REGION Network 52: Call CM Electrode Fix Left Top Up/Down (LBC_TwoWayActuator)
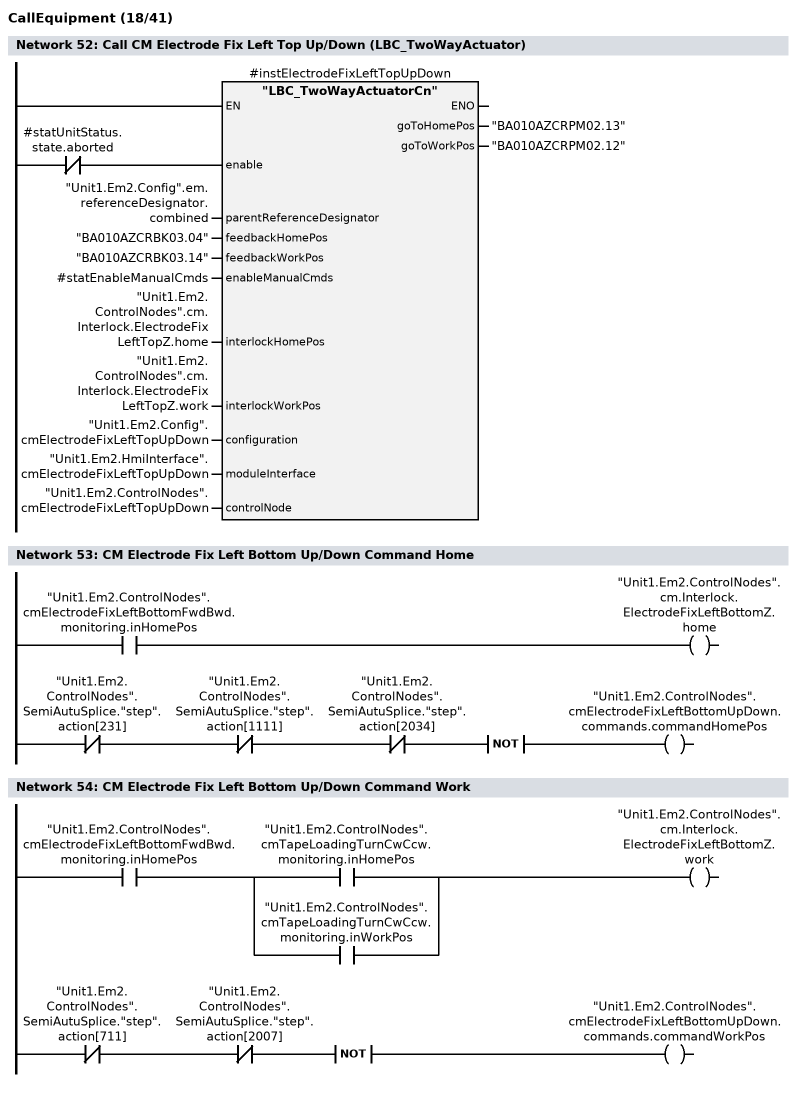
   RUNG wire#powerrail
      #instElectrodeFixLeftTopUpDown(enable := wire#w1, parentReferenceDesignator := "Unit1.Em2.Config".em.referenceDesignator.combined, feedbackHomePos := "BA010AZCRBK03.04", feedbackWorkPos := "BA010AZCRBK03.14", enableManualCmds := #statEnableManualCmds, interlockHomePos := "Unit1.Em2.ControlNodes".cm.Interlock.ElectrodeFixLeftTopZ.home, interlockWorkPos := "Unit1.Em2.ControlNodes".cm.Interlock.ElectrodeFixLeftTopZ.work, configuration := "Unit1.Em2.Config".cmElectrodeFixLeftTopUpDown, moduleInterface := "Unit1.Em2.HmiInterface".cmElectrodeFixLeftTopUpDown, controlNode := "Unit1.Em2.ControlNodes".cmElectrodeFixLeftTopUpDown, goToHomePos => "BA010AZCRPM02.13", goToWorkPos => "BA010AZCRPM02.12")
   END_RUNG
   RUNG wire#powerrail
      I_Contact( #statUnitStatus.state.aborted )
   END_RUNG wire#w1
   // the same network as SCL:
   #instElectrodeFixLeftTopUpDown(enable := NOT #statUnitStatus.state.aborted,   // "LBC_TwoWayActuatorCn"
                           parentReferenceDesignator := "Unit1.Em2.Config".em.referenceDesignator.combined,
                           feedbackHomePos := "BA010AZCRBK03.04",
                           feedbackWorkPos := "BA010AZCRBK03.14",
                           enableManualCmds := #statEnableManualCmds,
                           interlockHomePos := "Unit1.Em2.ControlNodes".cm.Interlock.ElectrodeFixLeftTopZ.home,
                           interlockWorkPos := "Unit1.Em2.ControlNodes".cm.Interlock.ElectrodeFixLeftTopZ.work,
                           configuration := "Unit1.Em2.Config".cmElectrodeFixLeftTopUpDown,
                           moduleInterface := "Unit1.Em2.HmiInterface".cmElectrodeFixLeftTopUpDown,
                           controlNode := "Unit1.Em2.ControlNodes".cmElectrodeFixLeftTopUpDown,
                           goToHomePos => "BA010AZCRPM02.13",
                           goToWorkPos => "BA010AZCRPM02.12");
END_REGION

REGION Network 53: CM Electrode Fix Left Bottom Up/Down Command Home
   RUNG wire#powerrail
      Contact( "Unit1.Em2.ControlNodes".cmElectrodeFixLeftBottomFwdBwd.monitoring.inHomePos )
      Coil( "Unit1.Em2.ControlNodes".cm.Interlock.ElectrodeFixLeftBottomZ.home )
   END_RUNG
   RUNG wire#powerrail
      I_Contact( "Unit1.Em2.ControlNodes".SemiAutuSplice."step".action[231] )
      I_Contact( "Unit1.Em2.ControlNodes".SemiAutuSplice."step".action[1111] )
      I_Contact( "Unit1.Em2.ControlNodes".SemiAutuSplice."step".action[2034] )
      Not()
      Coil( "Unit1.Em2.ControlNodes".cmElectrodeFixLeftBottomUpDown.commands.commandHomePos )
   END_RUNG
   // the same network as SCL:
   "Unit1.Em2.ControlNodes".cm.Interlock.ElectrodeFixLeftBottomZ.home := "Unit1.Em2.ControlNodes".cmElectrodeFixLeftBottomFwdBwd.monitoring.inHomePos;
   "Unit1.Em2.ControlNodes".cmElectrodeFixLeftBottomUpDown.commands.commandHomePos := NOT (NOT "Unit1.Em2.ControlNodes".SemiAutuSplice."step".action[231] AND NOT "Unit1.Em2.ControlNodes".SemiAutuSplice."step".action[1111] AND NOT "Unit1.Em2.ControlNodes".SemiAutuSplice."step".action[2034]);
END_REGION

REGION Network 54: CM Electrode Fix Left Bottom Up/Down Command Work
   RUNG wire#powerrail
      Contact( "Unit1.Em2.ControlNodes".cmElectrodeFixLeftBottomFwdBwd.monitoring.inHomePos )
      wire#w1
      Contact( "Unit1.Em2.ControlNodes".cmTapeLoadingTurnCwCcw.monitoring.inHomePos )
      wire#w2
      Coil( "Unit1.Em2.ControlNodes".cm.Interlock.ElectrodeFixLeftBottomZ.work )
   END_RUNG
   RUNG wire#w1
      Contact( "Unit1.Em2.ControlNodes".cmTapeLoadingTurnCwCcw.monitoring.inWorkPos )
   END_RUNG wire#w2
   RUNG wire#powerrail
      I_Contact( "Unit1.Em2.ControlNodes".SemiAutuSplice."step".action[711] )
      I_Contact( "Unit1.Em2.ControlNodes".SemiAutuSplice."step".action[2007] )
      Not()
      Coil( "Unit1.Em2.ControlNodes".cmElectrodeFixLeftBottomUpDown.commands.commandWorkPos )
   END_RUNG
   // the same network as SCL:
   "Unit1.Em2.ControlNodes".cm.Interlock.ElectrodeFixLeftBottomZ.work := "Unit1.Em2.ControlNodes".cmElectrodeFixLeftBottomFwdBwd.monitoring.inHomePos AND ("Unit1.Em2.ControlNodes".cmTapeLoadingTurnCwCcw.monitoring.inHomePos OR "Unit1.Em2.ControlNodes".cmTapeLoadingTurnCwCcw.monitoring.inWorkPos);
   "Unit1.Em2.ControlNodes".cmElectrodeFixLeftBottomUpDown.commands.commandWorkPos := NOT (NOT "Unit1.Em2.ControlNodes".SemiAutuSplice."step".action[711] AND NOT "Unit1.Em2.ControlNodes".SemiAutuSplice."step".action[2007]);
END_REGION

REGION Network 55: Call CM Electrode Fix Left Bottom Up/Down (LBC_TwoWayActuator)
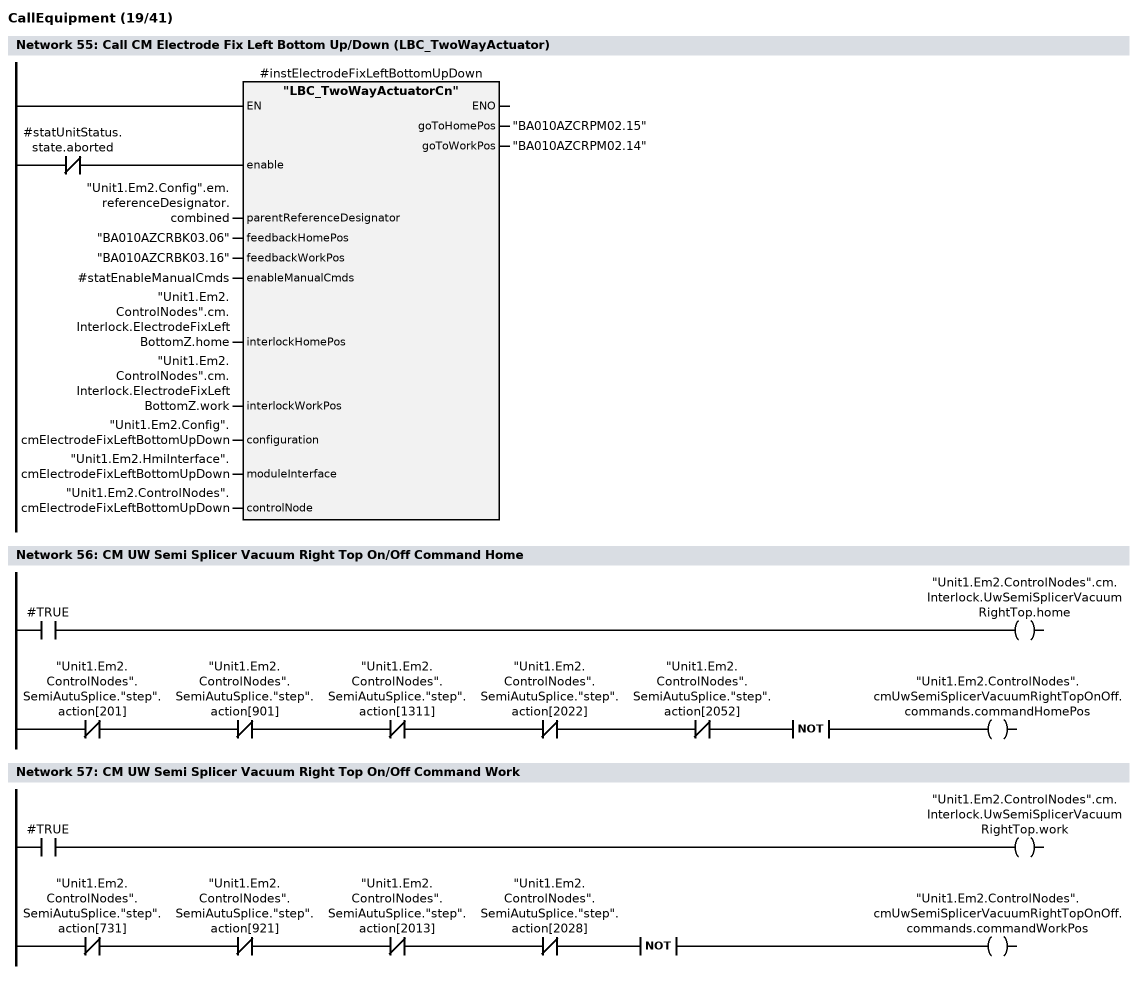
   RUNG wire#powerrail
      #instElectrodeFixLeftBottomUpDown(enable := wire#w1, parentReferenceDesignator := "Unit1.Em2.Config".em.referenceDesignator.combined, feedbackHomePos := "BA010AZCRBK03.06", feedbackWorkPos := "BA010AZCRBK03.16", enableManualCmds := #statEnableManualCmds, interlockHomePos := "Unit1.Em2.ControlNodes".cm.Interlock.ElectrodeFixLeftBottomZ.home, interlockWorkPos := "Unit1.Em2.ControlNodes".cm.Interlock.ElectrodeFixLeftBottomZ.work, configuration := "Unit1.Em2.Config".cmElectrodeFixLeftBottomUpDown, moduleInterface := "Unit1.Em2.HmiInterface".cmElectrodeFixLeftBottomUpDown, controlNode := "Unit1.Em2.ControlNodes".cmElectrodeFixLeftBottomUpDown, goToHomePos => "BA010AZCRPM02.15", goToWorkPos => "BA010AZCRPM02.14")
   END_RUNG
   RUNG wire#powerrail
      I_Contact( #statUnitStatus.state.aborted )
   END_RUNG wire#w1
   // the same network as SCL:
   #instElectrodeFixLeftBottomUpDown(enable := NOT #statUnitStatus.state.aborted,   // "LBC_TwoWayActuatorCn"
                           parentReferenceDesignator := "Unit1.Em2.Config".em.referenceDesignator.combined,
                           feedbackHomePos := "BA010AZCRBK03.06",
                           feedbackWorkPos := "BA010AZCRBK03.16",
                           enableManualCmds := #statEnableManualCmds,
                           interlockHomePos := "Unit1.Em2.ControlNodes".cm.Interlock.ElectrodeFixLeftBottomZ.home,
                           interlockWorkPos := "Unit1.Em2.ControlNodes".cm.Interlock.ElectrodeFixLeftBottomZ.work,
                           configuration := "Unit1.Em2.Config".cmElectrodeFixLeftBottomUpDown,
                           moduleInterface := "Unit1.Em2.HmiInterface".cmElectrodeFixLeftBottomUpDown,
                           controlNode := "Unit1.Em2.ControlNodes".cmElectrodeFixLeftBottomUpDown,
                           goToHomePos => "BA010AZCRPM02.15",
                           goToWorkPos => "BA010AZCRPM02.14");
END_REGION

REGION Network 56: CM UW Semi Splicer Vacuum Right Top On/Off Command Home
   RUNG wire#powerrail
      Contact( #TRUE )
      Coil( "Unit1.Em2.ControlNodes".cm.Interlock.UwSemiSplicerVacuumRightTop.home )
   END_RUNG
   RUNG wire#powerrail
      I_Contact( "Unit1.Em2.ControlNodes".SemiAutuSplice."step".action[201] )
      I_Contact( "Unit1.Em2.ControlNodes".SemiAutuSplice."step".action[901] )
      I_Contact( "Unit1.Em2.ControlNodes".SemiAutuSplice."step".action[1311] )
      I_Contact( "Unit1.Em2.ControlNodes".SemiAutuSplice."step".action[2022] )
      I_Contact( "Unit1.Em2.ControlNodes".SemiAutuSplice."step".action[2052] )
      Not()
      Coil( "Unit1.Em2.ControlNodes".cmUwSemiSplicerVacuumRightTopOnOff.commands.commandHomePos )
   END_RUNG
   // the same network as SCL:
   "Unit1.Em2.ControlNodes".cm.Interlock.UwSemiSplicerVacuumRightTop.home := #TRUE;
   "Unit1.Em2.ControlNodes".cmUwSemiSplicerVacuumRightTopOnOff.commands.commandHomePos := NOT (NOT "Unit1.Em2.ControlNodes".SemiAutuSplice."step".action[201] AND NOT "Unit1.Em2.ControlNodes".SemiAutuSplice."step".action[901] AND NOT "Unit1.Em2.ControlNodes".SemiAutuSplice."step".action[1311] AND NOT "Unit1.Em2.ControlNodes".SemiAutuSplice."step".action[2022] AND NOT "Unit1.Em2.ControlNodes".SemiAutuSplice."step".action[2052]);
END_REGION

REGION Network 57: CM UW Semi Splicer Vacuum Right Top On/Off Command Work
   RUNG wire#powerrail
      Contact( #TRUE )
      Coil( "Unit1.Em2.ControlNodes".cm.Interlock.UwSemiSplicerVacuumRightTop.work )
   END_RUNG
   RUNG wire#powerrail
      I_Contact( "Unit1.Em2.ControlNodes".SemiAutuSplice."step".action[731] )
      I_Contact( "Unit1.Em2.ControlNodes".SemiAutuSplice."step".action[921] )
      I_Contact( "Unit1.Em2.ControlNodes".SemiAutuSplice."step".action[2013] )
      I_Contact( "Unit1.Em2.ControlNodes".SemiAutuSplice."step".action[2028] )
      Not()
      Coil( "Unit1.Em2.ControlNodes".cmUwSemiSplicerVacuumRightTopOnOff.commands.commandWorkPos )
   END_RUNG
   // the same network as SCL:
   "Unit1.Em2.ControlNodes".cm.Interlock.UwSemiSplicerVacuumRightTop.work := #TRUE;
   "Unit1.Em2.ControlNodes".cmUwSemiSplicerVacuumRightTopOnOff.commands.commandWorkPos := NOT (NOT "Unit1.Em2.ControlNodes".SemiAutuSplice."step".action[731] AND NOT "Unit1.Em2.ControlNodes".SemiAutuSplice."step".action[921] AND NOT "Unit1.Em2.ControlNodes".SemiAutuSplice."step".action[2013] AND NOT "Unit1.Em2.ControlNodes".SemiAutuSplice."step".action[2028]);
END_REGION

REGION Network 58: Call CM UW Semi Splicer Vacuum Right Top On/Off (LBC_TwoWayActuator)
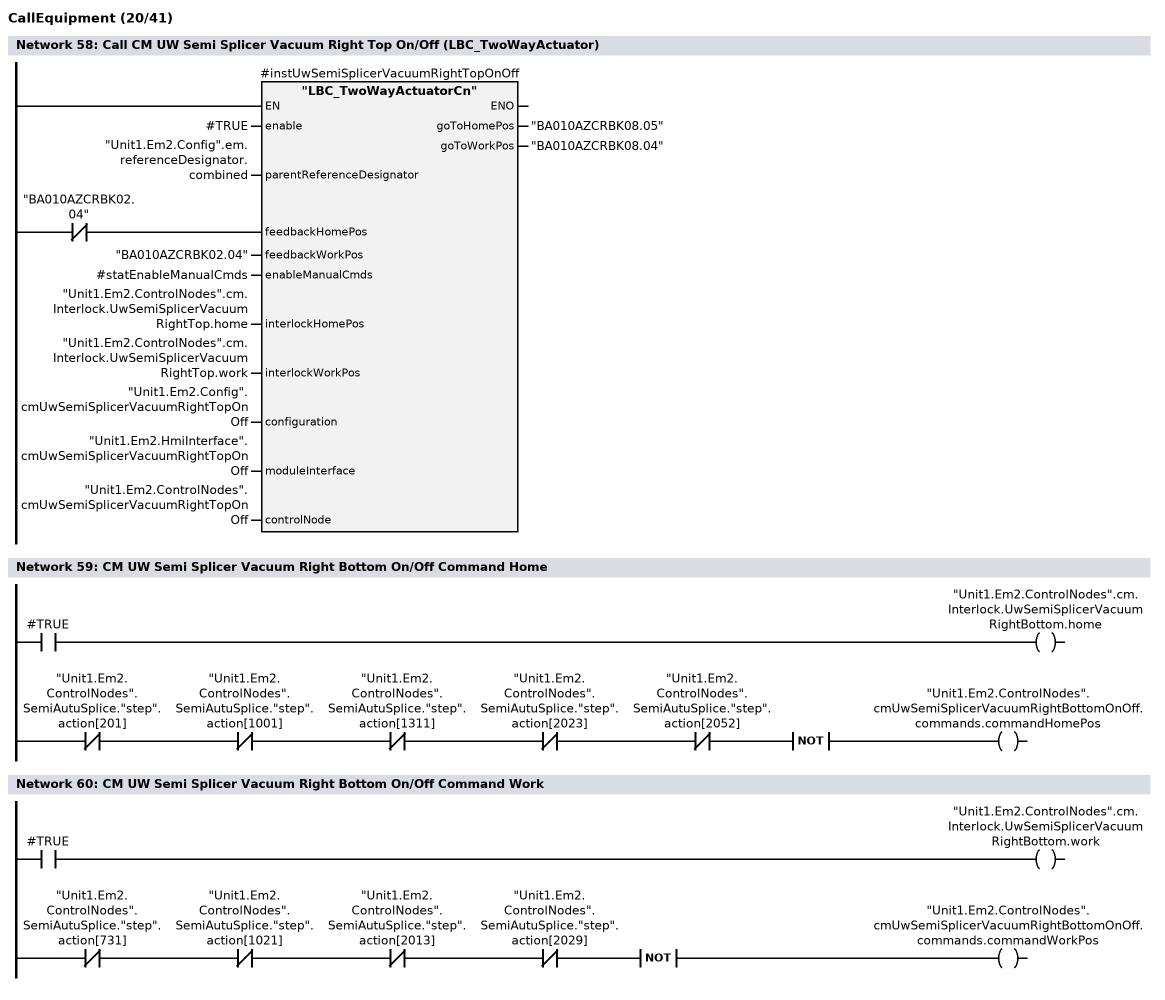
   RUNG wire#powerrail
      #instUwSemiSplicerVacuumRightTopOnOff(feedbackHomePos := wire#w1, enable := #TRUE, parentReferenceDesignator := "Unit1.Em2.Config".em.referenceDesignator.combined, feedbackWorkPos := "BA010AZCRBK02.04", enableManualCmds := #statEnableManualCmds, interlockHomePos := "Unit1.Em2.ControlNodes".cm.Interlock.UwSemiSplicerVacuumRightTop.home, interlockWorkPos := "Unit1.Em2.ControlNodes".cm.Interlock.UwSemiSplicerVacuumRightTop.work, configuration := "Unit1.Em2.Config".cmUwSemiSplicerVacuumRightTopOnOff, moduleInterface := "Unit1.Em2.HmiInterface".cmUwSemiSplicerVacuumRightTopOnOff, controlNode := "Unit1.Em2.ControlNodes".cmUwSemiSplicerVacuumRightTopOnOff, goToHomePos => "BA010AZCRBK08.05", goToWorkPos => "BA010AZCRBK08.04")
   END_RUNG
   RUNG wire#powerrail
      I_Contact( "BA010AZCRBK02.04" )
   END_RUNG wire#w1
   // the same network as SCL:
   #instUwSemiSplicerVacuumRightTopOnOff(enable := #TRUE,   // "LBC_TwoWayActuatorCn"
                           parentReferenceDesignator := "Unit1.Em2.Config".em.referenceDesignator.combined,
                           feedbackHomePos := NOT "BA010AZCRBK02.04",
                           feedbackWorkPos := "BA010AZCRBK02.04",
                           enableManualCmds := #statEnableManualCmds,
                           interlockHomePos := "Unit1.Em2.ControlNodes".cm.Interlock.UwSemiSplicerVacuumRightTop.home,
                           interlockWorkPos := "Unit1.Em2.ControlNodes".cm.Interlock.UwSemiSplicerVacuumRightTop.work,
                           configuration := "Unit1.Em2.Config".cmUwSemiSplicerVacuumRightTopOnOff,
                           moduleInterface := "Unit1.Em2.HmiInterface".cmUwSemiSplicerVacuumRightTopOnOff,
                           controlNode := "Unit1.Em2.ControlNodes".cmUwSemiSplicerVacuumRightTopOnOff,
                           goToHomePos => "BA010AZCRBK08.05",
                           goToWorkPos => "BA010AZCRBK08.04");
END_REGION

REGION Network 59: CM UW Semi Splicer Vacuum Right Bottom On/Off Command Home
   RUNG wire#powerrail
      Contact( #TRUE )
      Coil( "Unit1.Em2.ControlNodes".cm.Interlock.UwSemiSplicerVacuumRightBottom.home )
   END_RUNG
   RUNG wire#powerrail
      I_Contact( "Unit1.Em2.ControlNodes".SemiAutuSplice."step".action[201] )
      I_Contact( "Unit1.Em2.ControlNodes".SemiAutuSplice."step".action[1001] )
      I_Contact( "Unit1.Em2.ControlNodes".SemiAutuSplice."step".action[1311] )
      I_Contact( "Unit1.Em2.ControlNodes".SemiAutuSplice."step".action[2023] )
      I_Contact( "Unit1.Em2.ControlNodes".SemiAutuSplice."step".action[2052] )
      Not()
      Coil( "Unit1.Em2.ControlNodes".cmUwSemiSplicerVacuumRightBottomOnOff.commands.commandHomePos )
   END_RUNG
   // the same network as SCL:
   "Unit1.Em2.ControlNodes".cm.Interlock.UwSemiSplicerVacuumRightBottom.home := #TRUE;
   "Unit1.Em2.ControlNodes".cmUwSemiSplicerVacuumRightBottomOnOff.commands.commandHomePos := NOT (NOT "Unit1.Em2.ControlNodes".SemiAutuSplice."step".action[201] AND NOT "Unit1.Em2.ControlNodes".SemiAutuSplice."step".action[1001] AND NOT "Unit1.Em2.ControlNodes".SemiAutuSplice."step".action[1311] AND NOT "Unit1.Em2.ControlNodes".SemiAutuSplice."step".action[2023] AND NOT "Unit1.Em2.ControlNodes".SemiAutuSplice."step".action[2052]);
END_REGION

REGION Network 60: CM UW Semi Splicer Vacuum Right Bottom On/Off Command Work
   RUNG wire#powerrail
      Contact( #TRUE )
      Coil( "Unit1.Em2.ControlNodes".cm.Interlock.UwSemiSplicerVacuumRightBottom.work )
   END_RUNG
   RUNG wire#powerrail
      I_Contact( "Unit1.Em2.ControlNodes".SemiAutuSplice."step".action[731] )
      I_Contact( "Unit1.Em2.ControlNodes".SemiAutuSplice."step".action[1021] )
      I_Contact( "Unit1.Em2.ControlNodes".SemiAutuSplice."step".action[2013] )
      I_Contact( "Unit1.Em2.ControlNodes".SemiAutuSplice."step".action[2029] )
      Not()
      Coil( "Unit1.Em2.ControlNodes".cmUwSemiSplicerVacuumRightBottomOnOff.commands.commandWorkPos )
   END_RUNG
   // the same network as SCL:
   "Unit1.Em2.ControlNodes".cm.Interlock.UwSemiSplicerVacuumRightBottom.work := #TRUE;
   "Unit1.Em2.ControlNodes".cmUwSemiSplicerVacuumRightBottomOnOff.commands.commandWorkPos := NOT (NOT "Unit1.Em2.ControlNodes".SemiAutuSplice."step".action[731] AND NOT "Unit1.Em2.ControlNodes".SemiAutuSplice."step".action[1021] AND NOT "Unit1.Em2.ControlNodes".SemiAutuSplice."step".action[2013] AND NOT "Unit1.Em2.ControlNodes".SemiAutuSplice."step".action[2029]);
END_REGION

REGION Network 61: Call CM UW Semi Splicer Vacuum Right Bottom On/Off (LBC_TwoWayActuator)
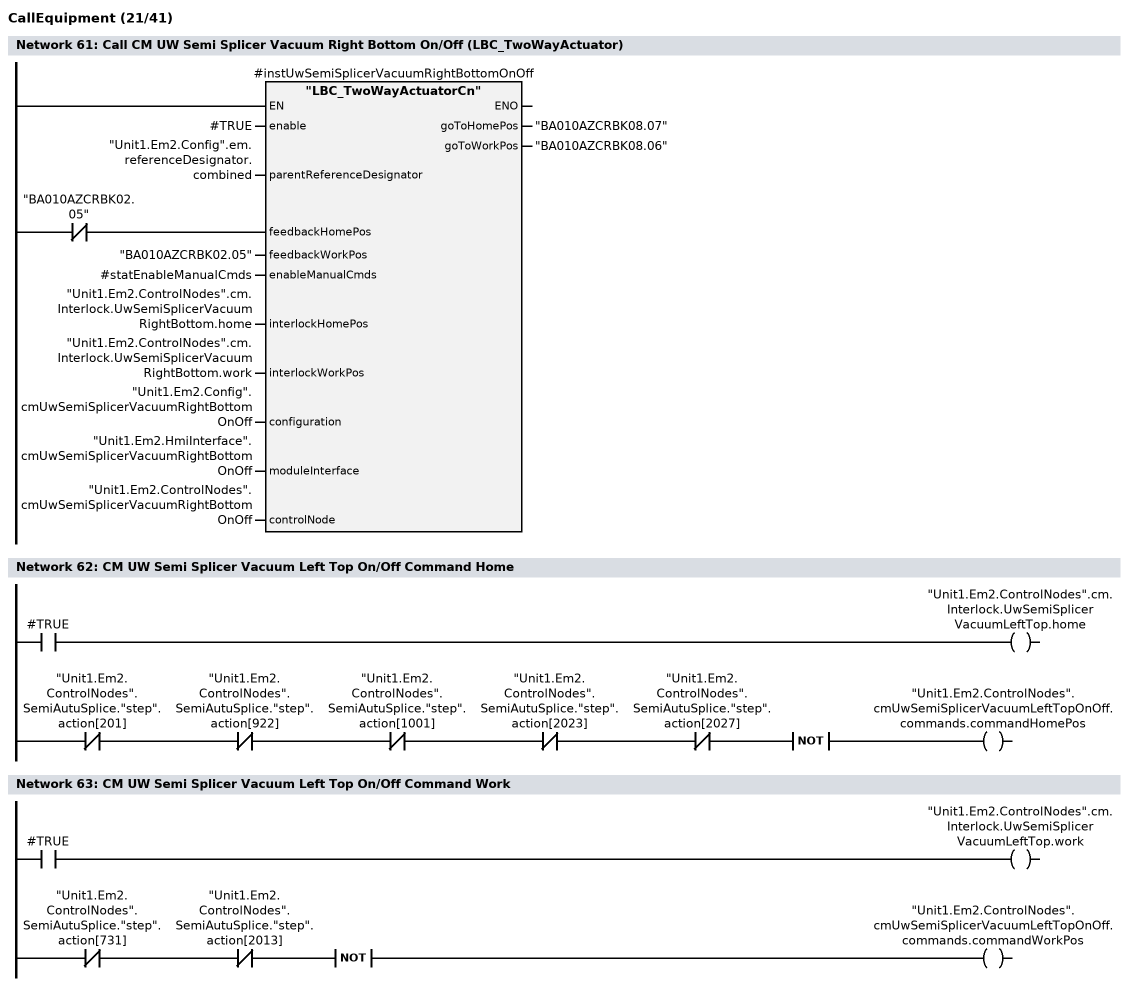
   RUNG wire#powerrail
      #instUwSemiSplicerVacuumRightBottomOnOff(feedbackHomePos := wire#w1, enable := #TRUE, parentReferenceDesignator := "Unit1.Em2.Config".em.referenceDesignator.combined, feedbackWorkPos := "BA010AZCRBK02.05", enableManualCmds := #statEnableManualCmds, interlockHomePos := "Unit1.Em2.ControlNodes".cm.Interlock.UwSemiSplicerVacuumRightBottom.home, interlockWorkPos := "Unit1.Em2.ControlNodes".cm.Interlock.UwSemiSplicerVacuumRightBottom.work, configuration := "Unit1.Em2.Config".cmUwSemiSplicerVacuumRightBottomOnOff, moduleInterface := "Unit1.Em2.HmiInterface".cmUwSemiSplicerVacuumRightBottomOnOff, controlNode := "Unit1.Em2.ControlNodes".cmUwSemiSplicerVacuumRightBottomOnOff, goToHomePos => "BA010AZCRBK08.07", goToWorkPos => "BA010AZCRBK08.06")
   END_RUNG
   RUNG wire#powerrail
      I_Contact( "BA010AZCRBK02.05" )
   END_RUNG wire#w1
   // the same network as SCL:
   #instUwSemiSplicerVacuumRightBottomOnOff(enable := #TRUE,   // "LBC_TwoWayActuatorCn"
                           parentReferenceDesignator := "Unit1.Em2.Config".em.referenceDesignator.combined,
                           feedbackHomePos := NOT "BA010AZCRBK02.05",
                           feedbackWorkPos := "BA010AZCRBK02.05",
                           enableManualCmds := #statEnableManualCmds,
                           interlockHomePos := "Unit1.Em2.ControlNodes".cm.Interlock.UwSemiSplicerVacuumRightBottom.home,
                           interlockWorkPos := "Unit1.Em2.ControlNodes".cm.Interlock.UwSemiSplicerVacuumRightBottom.work,
                           configuration := "Unit1.Em2.Config".cmUwSemiSplicerVacuumRightBottomOnOff,
                           moduleInterface := "Unit1.Em2.HmiInterface".cmUwSemiSplicerVacuumRightBottomOnOff,
                           controlNode := "Unit1.Em2.ControlNodes".cmUwSemiSplicerVacuumRightBottomOnOff,
                           goToHomePos => "BA010AZCRBK08.07",
                           goToWorkPos => "BA010AZCRBK08.06");
END_REGION

REGION Network 62: CM UW Semi Splicer Vacuum Left Top On/Off Command Home
   RUNG wire#powerrail
      Contact( #TRUE )
      Coil( "Unit1.Em2.ControlNodes".cm.Interlock.UwSemiSplicerVacuumLeftTop.home )
   END_RUNG
   RUNG wire#powerrail
      I_Contact( "Unit1.Em2.ControlNodes".SemiAutuSplice."step".action[201] )
      I_Contact( "Unit1.Em2.ControlNodes".SemiAutuSplice."step".action[922] )
      I_Contact( "Unit1.Em2.ControlNodes".SemiAutuSplice."step".action[1001] )
      I_Contact( "Unit1.Em2.ControlNodes".SemiAutuSplice."step".action[2023] )
      I_Contact( "Unit1.Em2.ControlNodes".SemiAutuSplice."step".action[2027] )
      Not()
      Coil( "Unit1.Em2.ControlNodes".cmUwSemiSplicerVacuumLeftTopOnOff.commands.commandHomePos )
   END_RUNG
   // the same network as SCL:
   "Unit1.Em2.ControlNodes".cm.Interlock.UwSemiSplicerVacuumLeftTop.home := #TRUE;
   "Unit1.Em2.ControlNodes".cmUwSemiSplicerVacuumLeftTopOnOff.commands.commandHomePos := NOT (NOT "Unit1.Em2.ControlNodes".SemiAutuSplice."step".action[201] AND NOT "Unit1.Em2.ControlNodes".SemiAutuSplice."step".action[922] AND NOT "Unit1.Em2.ControlNodes".SemiAutuSplice."step".action[1001] AND NOT "Unit1.Em2.ControlNodes".SemiAutuSplice."step".action[2023] AND NOT "Unit1.Em2.ControlNodes".SemiAutuSplice."step".action[2027]);
END_REGION

REGION Network 63: CM UW Semi Splicer Vacuum Left Top On/Off Command Work
   RUNG wire#powerrail
      Contact( #TRUE )
      Coil( "Unit1.Em2.ControlNodes".cm.Interlock.UwSemiSplicerVacuumLeftTop.work )
   END_RUNG
   RUNG wire#powerrail
      I_Contact( "Unit1.Em2.ControlNodes".SemiAutuSplice."step".action[731] )
      I_Contact( "Unit1.Em2.ControlNodes".SemiAutuSplice."step".action[2013] )
      Not()
      Coil( "Unit1.Em2.ControlNodes".cmUwSemiSplicerVacuumLeftTopOnOff.commands.commandWorkPos )
   END_RUNG
   // the same network as SCL:
   "Unit1.Em2.ControlNodes".cm.Interlock.UwSemiSplicerVacuumLeftTop.work := #TRUE;
   "Unit1.Em2.ControlNodes".cmUwSemiSplicerVacuumLeftTopOnOff.commands.commandWorkPos := NOT (NOT "Unit1.Em2.ControlNodes".SemiAutuSplice."step".action[731] AND NOT "Unit1.Em2.ControlNodes".SemiAutuSplice."step".action[2013]);
END_REGION

REGION Network 64: Call CM UW Semi Splicer Vacuum Left Top On/Off (LBC_TwoWayActuator)
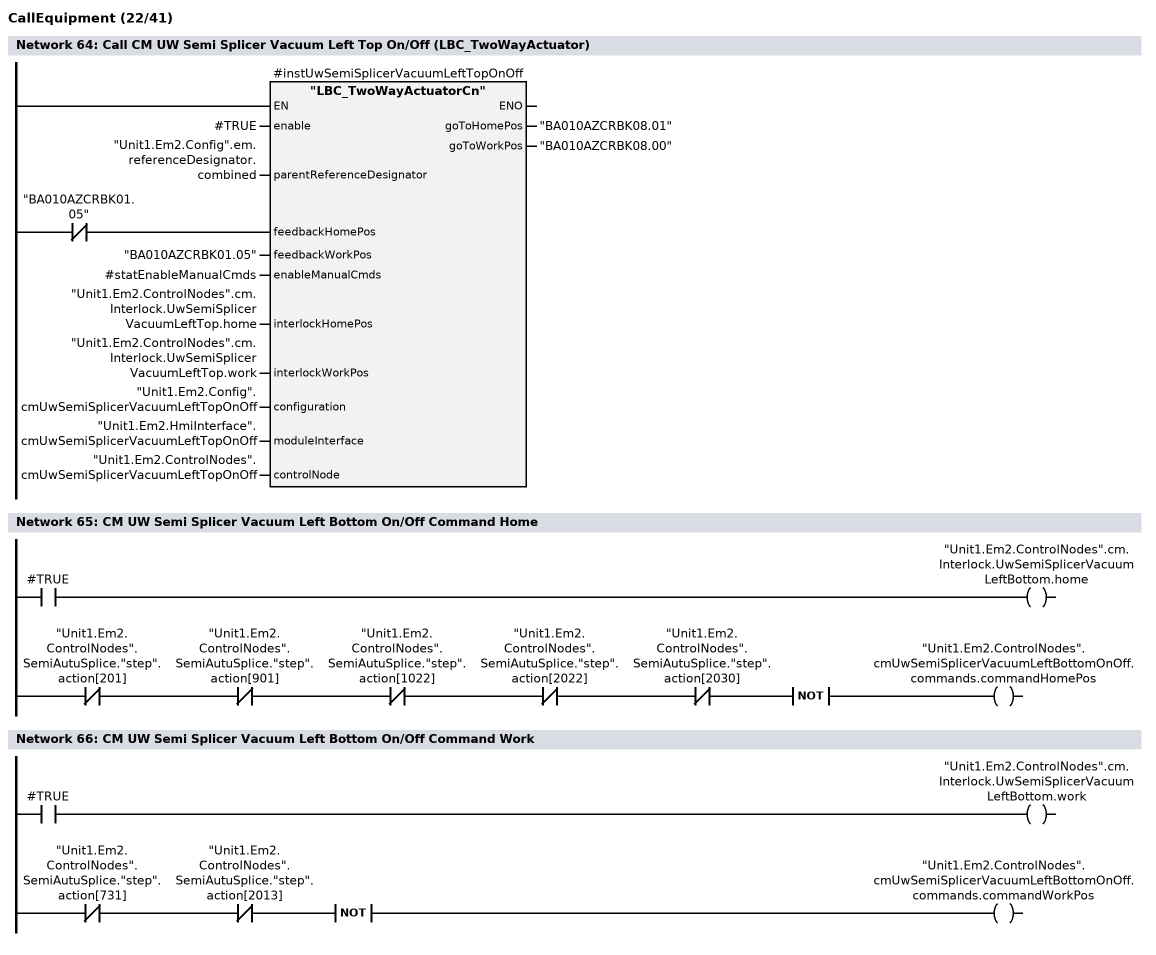
   RUNG wire#powerrail
      #instUwSemiSplicerVacuumLeftTopOnOff(feedbackHomePos := wire#w1, enable := #TRUE, parentReferenceDesignator := "Unit1.Em2.Config".em.referenceDesignator.combined, feedbackWorkPos := "BA010AZCRBK01.05", enableManualCmds := #statEnableManualCmds, interlockHomePos := "Unit1.Em2.ControlNodes".cm.Interlock.UwSemiSplicerVacuumLeftTop.home, interlockWorkPos := "Unit1.Em2.ControlNodes".cm.Interlock.UwSemiSplicerVacuumLeftTop.work, configuration := "Unit1.Em2.Config".cmUwSemiSplicerVacuumLeftTopOnOff, moduleInterface := "Unit1.Em2.HmiInterface".cmUwSemiSplicerVacuumLeftTopOnOff, controlNode := "Unit1.Em2.ControlNodes".cmUwSemiSplicerVacuumLeftTopOnOff, goToHomePos => "BA010AZCRBK08.01", goToWorkPos => "BA010AZCRBK08.00")
   END_RUNG
   RUNG wire#powerrail
      I_Contact( "BA010AZCRBK01.05" )
   END_RUNG wire#w1
   // the same network as SCL:
   #instUwSemiSplicerVacuumLeftTopOnOff(enable := #TRUE,   // "LBC_TwoWayActuatorCn"
                           parentReferenceDesignator := "Unit1.Em2.Config".em.referenceDesignator.combined,
                           feedbackHomePos := NOT "BA010AZCRBK01.05",
                           feedbackWorkPos := "BA010AZCRBK01.05",
                           enableManualCmds := #statEnableManualCmds,
                           interlockHomePos := "Unit1.Em2.ControlNodes".cm.Interlock.UwSemiSplicerVacuumLeftTop.home,
                           interlockWorkPos := "Unit1.Em2.ControlNodes".cm.Interlock.UwSemiSplicerVacuumLeftTop.work,
                           configuration := "Unit1.Em2.Config".cmUwSemiSplicerVacuumLeftTopOnOff,
                           moduleInterface := "Unit1.Em2.HmiInterface".cmUwSemiSplicerVacuumLeftTopOnOff,
                           controlNode := "Unit1.Em2.ControlNodes".cmUwSemiSplicerVacuumLeftTopOnOff,
                           goToHomePos => "BA010AZCRBK08.01",
                           goToWorkPos => "BA010AZCRBK08.00");
END_REGION

REGION Network 65: CM UW Semi Splicer Vacuum Left Bottom On/Off Command Home
   RUNG wire#powerrail
      Contact( #TRUE )
      Coil( "Unit1.Em2.ControlNodes".cm.Interlock.UwSemiSplicerVacuumLeftBottom.home )
   END_RUNG
   RUNG wire#powerrail
      I_Contact( "Unit1.Em2.ControlNodes".SemiAutuSplice."step".action[201] )
      I_Contact( "Unit1.Em2.ControlNodes".SemiAutuSplice."step".action[901] )
      I_Contact( "Unit1.Em2.ControlNodes".SemiAutuSplice."step".action[1022] )
      I_Contact( "Unit1.Em2.ControlNodes".SemiAutuSplice."step".action[2022] )
      I_Contact( "Unit1.Em2.ControlNodes".SemiAutuSplice."step".action[2030] )
      Not()
      Coil( "Unit1.Em2.ControlNodes".cmUwSemiSplicerVacuumLeftBottomOnOff.commands.commandHomePos )
   END_RUNG
   // the same network as SCL:
   "Unit1.Em2.ControlNodes".cm.Interlock.UwSemiSplicerVacuumLeftBottom.home := #TRUE;
   "Unit1.Em2.ControlNodes".cmUwSemiSplicerVacuumLeftBottomOnOff.commands.commandHomePos := NOT (NOT "Unit1.Em2.ControlNodes".SemiAutuSplice."step".action[201] AND NOT "Unit1.Em2.ControlNodes".SemiAutuSplice."step".action[901] AND NOT "Unit1.Em2.ControlNodes".SemiAutuSplice."step".action[1022] AND NOT "Unit1.Em2.ControlNodes".SemiAutuSplice."step".action[2022] AND NOT "Unit1.Em2.ControlNodes".SemiAutuSplice."step".action[2030]);
END_REGION

REGION Network 66: CM UW Semi Splicer Vacuum Left Bottom On/Off Command Work
   RUNG wire#powerrail
      Contact( #TRUE )
      Coil( "Unit1.Em2.ControlNodes".cm.Interlock.UwSemiSplicerVacuumLeftBottom.work )
   END_RUNG
   RUNG wire#powerrail
      I_Contact( "Unit1.Em2.ControlNodes".SemiAutuSplice."step".action[731] )
      I_Contact( "Unit1.Em2.ControlNodes".SemiAutuSplice."step".action[2013] )
      Not()
      Coil( "Unit1.Em2.ControlNodes".cmUwSemiSplicerVacuumLeftBottomOnOff.commands.commandWorkPos )
   END_RUNG
   // the same network as SCL:
   "Unit1.Em2.ControlNodes".cm.Interlock.UwSemiSplicerVacuumLeftBottom.work := #TRUE;
   "Unit1.Em2.ControlNodes".cmUwSemiSplicerVacuumLeftBottomOnOff.commands.commandWorkPos := NOT (NOT "Unit1.Em2.ControlNodes".SemiAutuSplice."step".action[731] AND NOT "Unit1.Em2.ControlNodes".SemiAutuSplice."step".action[2013]);
END_REGION

REGION Network 67: Call CM UW Semi Splicer Vacuum Left Bottom On/Off (LBC_TwoWayActuator)
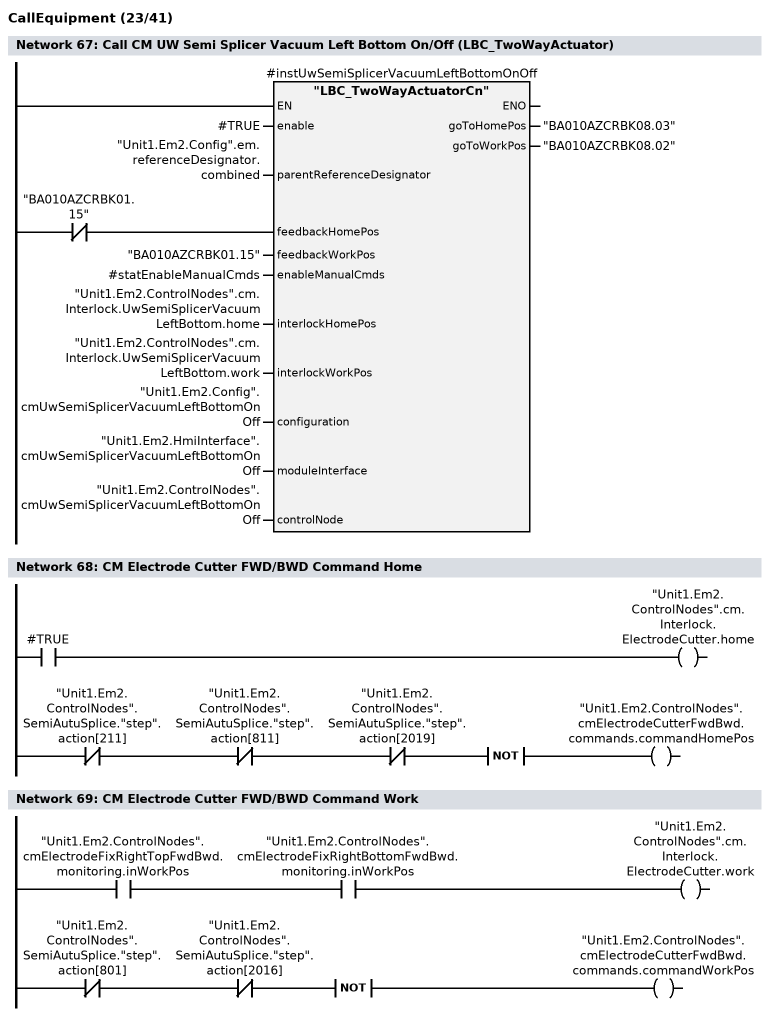
   RUNG wire#powerrail
      #instUwSemiSplicerVacuumLeftBottomOnOff(feedbackHomePos := wire#w1, enable := #TRUE, parentReferenceDesignator := "Unit1.Em2.Config".em.referenceDesignator.combined, feedbackWorkPos := "BA010AZCRBK01.15", enableManualCmds := #statEnableManualCmds, interlockHomePos := "Unit1.Em2.ControlNodes".cm.Interlock.UwSemiSplicerVacuumLeftBottom.home, interlockWorkPos := "Unit1.Em2.ControlNodes".cm.Interlock.UwSemiSplicerVacuumLeftBottom.work, configuration := "Unit1.Em2.Config".cmUwSemiSplicerVacuumLeftBottomOnOff, moduleInterface := "Unit1.Em2.HmiInterface".cmUwSemiSplicerVacuumLeftBottomOnOff, controlNode := "Unit1.Em2.ControlNodes".cmUwSemiSplicerVacuumLeftBottomOnOff, goToHomePos => "BA010AZCRBK08.03", goToWorkPos => "BA010AZCRBK08.02")
   END_RUNG
   RUNG wire#powerrail
      I_Contact( "BA010AZCRBK01.15" )
   END_RUNG wire#w1
   // the same network as SCL:
   #instUwSemiSplicerVacuumLeftBottomOnOff(enable := #TRUE,   // "LBC_TwoWayActuatorCn"
                           parentReferenceDesignator := "Unit1.Em2.Config".em.referenceDesignator.combined,
                           feedbackHomePos := NOT "BA010AZCRBK01.15",
                           feedbackWorkPos := "BA010AZCRBK01.15",
                           enableManualCmds := #statEnableManualCmds,
                           interlockHomePos := "Unit1.Em2.ControlNodes".cm.Interlock.UwSemiSplicerVacuumLeftBottom.home,
                           interlockWorkPos := "Unit1.Em2.ControlNodes".cm.Interlock.UwSemiSplicerVacuumLeftBottom.work,
                           configuration := "Unit1.Em2.Config".cmUwSemiSplicerVacuumLeftBottomOnOff,
                           moduleInterface := "Unit1.Em2.HmiInterface".cmUwSemiSplicerVacuumLeftBottomOnOff,
                           controlNode := "Unit1.Em2.ControlNodes".cmUwSemiSplicerVacuumLeftBottomOnOff,
                           goToHomePos => "BA010AZCRBK08.03",
                           goToWorkPos => "BA010AZCRBK08.02");
END_REGION

REGION Network 68: CM Electrode Cutter FWD/BWD Command Home
   RUNG wire#powerrail
      Contact( #TRUE )
      Coil( "Unit1.Em2.ControlNodes".cm.Interlock.ElectrodeCutter.home )
   END_RUNG
   RUNG wire#powerrail
      I_Contact( "Unit1.Em2.ControlNodes".SemiAutuSplice."step".action[211] )
      I_Contact( "Unit1.Em2.ControlNodes".SemiAutuSplice."step".action[811] )
      I_Contact( "Unit1.Em2.ControlNodes".SemiAutuSplice."step".action[2019] )
      Not()
      Coil( "Unit1.Em2.ControlNodes".cmElectrodeCutterFwdBwd.commands.commandHomePos )
   END_RUNG
   // the same network as SCL:
   "Unit1.Em2.ControlNodes".cm.Interlock.ElectrodeCutter.home := #TRUE;
   "Unit1.Em2.ControlNodes".cmElectrodeCutterFwdBwd.commands.commandHomePos := NOT (NOT "Unit1.Em2.ControlNodes".SemiAutuSplice."step".action[211] AND NOT "Unit1.Em2.ControlNodes".SemiAutuSplice."step".action[811] AND NOT "Unit1.Em2.ControlNodes".SemiAutuSplice."step".action[2019]);
END_REGION

REGION Network 69: CM Electrode Cutter FWD/BWD Command Work
   RUNG wire#powerrail
      Contact( "Unit1.Em2.ControlNodes".cmElectrodeFixRightTopFwdBwd.monitoring.inWorkPos )
      Contact( "Unit1.Em2.ControlNodes".cmElectrodeFixRightBottomFwdBwd.monitoring.inWorkPos )
      Coil( "Unit1.Em2.ControlNodes".cm.Interlock.ElectrodeCutter.work )
   END_RUNG
   RUNG wire#powerrail
      I_Contact( "Unit1.Em2.ControlNodes".SemiAutuSplice."step".action[801] )
      I_Contact( "Unit1.Em2.ControlNodes".SemiAutuSplice."step".action[2016] )
      Not()
      Coil( "Unit1.Em2.ControlNodes".cmElectrodeCutterFwdBwd.commands.commandWorkPos )
   END_RUNG
   // the same network as SCL:
   "Unit1.Em2.ControlNodes".cm.Interlock.ElectrodeCutter.work := "Unit1.Em2.ControlNodes".cmElectrodeFixRightTopFwdBwd.monitoring.inWorkPos AND "Unit1.Em2.ControlNodes".cmElectrodeFixRightBottomFwdBwd.monitoring.inWorkPos;
   "Unit1.Em2.ControlNodes".cmElectrodeCutterFwdBwd.commands.commandWorkPos := NOT (NOT "Unit1.Em2.ControlNodes".SemiAutuSplice."step".action[801] AND NOT "Unit1.Em2.ControlNodes".SemiAutuSplice."step".action[2016]);
END_REGION

REGION Network 70: Call CM Electrode Cutter FWD/BWD (LBC_TwoWayActuator)
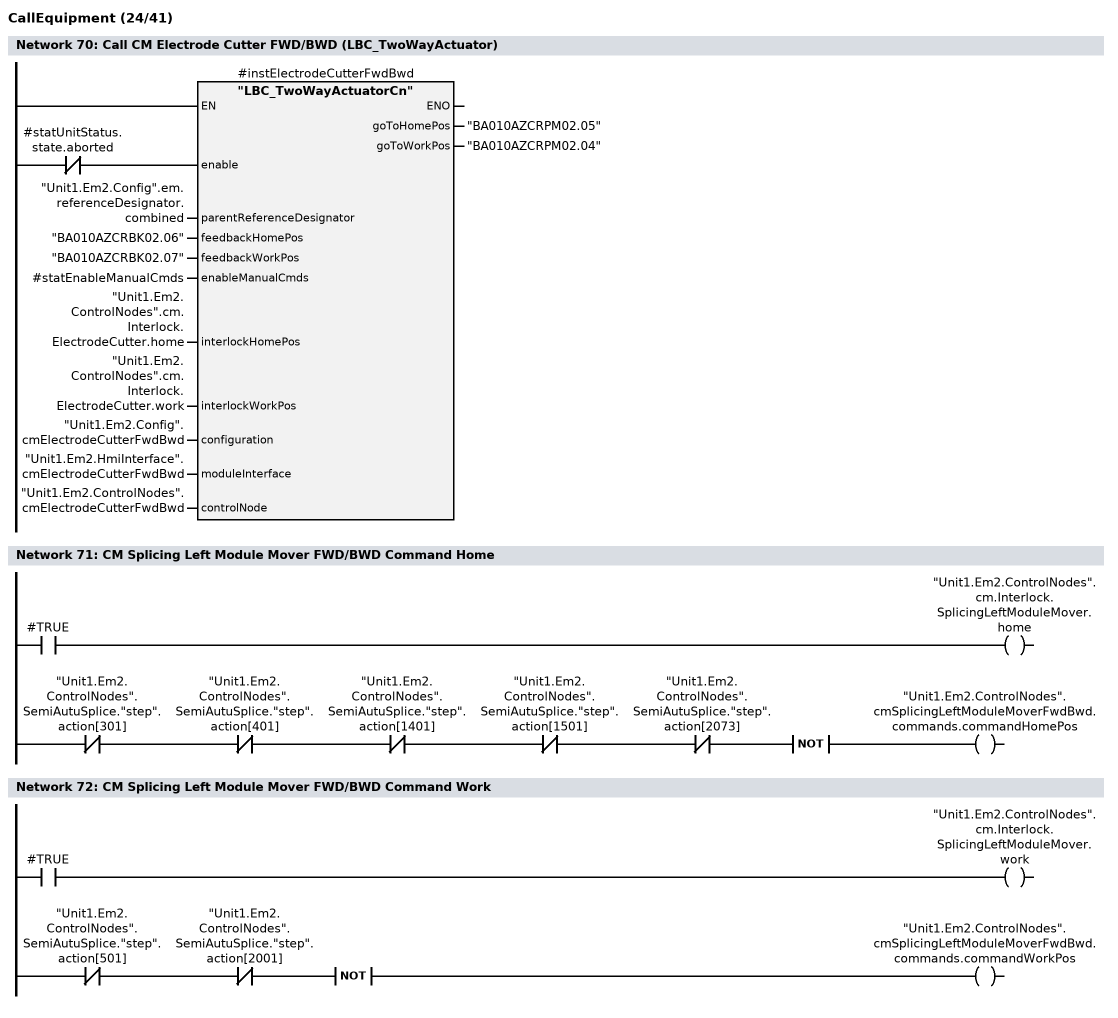
   RUNG wire#powerrail
      #instElectrodeCutterFwdBwd(enable := wire#w1, parentReferenceDesignator := "Unit1.Em2.Config".em.referenceDesignator.combined, feedbackHomePos := "BA010AZCRBK02.06", feedbackWorkPos := "BA010AZCRBK02.07", enableManualCmds := #statEnableManualCmds, interlockHomePos := "Unit1.Em2.ControlNodes".cm.Interlock.ElectrodeCutter.home, interlockWorkPos := "Unit1.Em2.ControlNodes".cm.Interlock.ElectrodeCutter.work, configuration := "Unit1.Em2.Config".cmElectrodeCutterFwdBwd, moduleInterface := "Unit1.Em2.HmiInterface".cmElectrodeCutterFwdBwd, controlNode := "Unit1.Em2.ControlNodes".cmElectrodeCutterFwdBwd, goToHomePos => "BA010AZCRPM02.05", goToWorkPos => "BA010AZCRPM02.04")
   END_RUNG
   RUNG wire#powerrail
      I_Contact( #statUnitStatus.state.aborted )
   END_RUNG wire#w1
   // the same network as SCL:
   #instElectrodeCutterFwdBwd(enable := NOT #statUnitStatus.state.aborted,   // "LBC_TwoWayActuatorCn"
                           parentReferenceDesignator := "Unit1.Em2.Config".em.referenceDesignator.combined,
                           feedbackHomePos := "BA010AZCRBK02.06",
                           feedbackWorkPos := "BA010AZCRBK02.07",
                           enableManualCmds := #statEnableManualCmds,
                           interlockHomePos := "Unit1.Em2.ControlNodes".cm.Interlock.ElectrodeCutter.home,
                           interlockWorkPos := "Unit1.Em2.ControlNodes".cm.Interlock.ElectrodeCutter.work,
                           configuration := "Unit1.Em2.Config".cmElectrodeCutterFwdBwd,
                           moduleInterface := "Unit1.Em2.HmiInterface".cmElectrodeCutterFwdBwd,
                           controlNode := "Unit1.Em2.ControlNodes".cmElectrodeCutterFwdBwd,
                           goToHomePos => "BA010AZCRPM02.05",
                           goToWorkPos => "BA010AZCRPM02.04");
END_REGION

REGION Network 71: CM Splicing Left Module Mover FWD/BWD Command Home
   RUNG wire#powerrail
      Contact( #TRUE )
      Coil( "Unit1.Em2.ControlNodes".cm.Interlock.SplicingLeftModuleMover.home )
   END_RUNG
   RUNG wire#powerrail
      I_Contact( "Unit1.Em2.ControlNodes".SemiAutuSplice."step".action[301] )
      I_Contact( "Unit1.Em2.ControlNodes".SemiAutuSplice."step".action[401] )
      I_Contact( "Unit1.Em2.ControlNodes".SemiAutuSplice."step".action[1401] )
      I_Contact( "Unit1.Em2.ControlNodes".SemiAutuSplice."step".action[1501] )
      I_Contact( "Unit1.Em2.ControlNodes".SemiAutuSplice."step".action[2073] )
      Not()
      Coil( "Unit1.Em2.ControlNodes".cmSplicingLeftModuleMoverFwdBwd.commands.commandHomePos )
   END_RUNG
   // the same network as SCL:
   "Unit1.Em2.ControlNodes".cm.Interlock.SplicingLeftModuleMover.home := #TRUE;
   "Unit1.Em2.ControlNodes".cmSplicingLeftModuleMoverFwdBwd.commands.commandHomePos := NOT (NOT "Unit1.Em2.ControlNodes".SemiAutuSplice."step".action[301] AND NOT "Unit1.Em2.ControlNodes".SemiAutuSplice."step".action[401] AND NOT "Unit1.Em2.ControlNodes".SemiAutuSplice."step".action[1401] AND NOT "Unit1.Em2.ControlNodes".SemiAutuSplice."step".action[1501] AND NOT "Unit1.Em2.ControlNodes".SemiAutuSplice."step".action[2073]);
END_REGION

REGION Network 72: CM Splicing Left Module Mover FWD/BWD Command Work
   RUNG wire#powerrail
      Contact( #TRUE )
      Coil( "Unit1.Em2.ControlNodes".cm.Interlock.SplicingLeftModuleMover.work )
   END_RUNG
   RUNG wire#powerrail
      I_Contact( "Unit1.Em2.ControlNodes".SemiAutuSplice."step".action[501] )
      I_Contact( "Unit1.Em2.ControlNodes".SemiAutuSplice."step".action[2001] )
      Not()
      Coil( "Unit1.Em2.ControlNodes".cmSplicingLeftModuleMoverFwdBwd.commands.commandWorkPos )
   END_RUNG
   // the same network as SCL:
   "Unit1.Em2.ControlNodes".cm.Interlock.SplicingLeftModuleMover.work := #TRUE;
   "Unit1.Em2.ControlNodes".cmSplicingLeftModuleMoverFwdBwd.commands.commandWorkPos := NOT (NOT "Unit1.Em2.ControlNodes".SemiAutuSplice."step".action[501] AND NOT "Unit1.Em2.ControlNodes".SemiAutuSplice."step".action[2001]);
END_REGION

REGION Network 73: Call CM Splicing Left Module Mover FWD/BWD (LBC_TwoWayActuator)
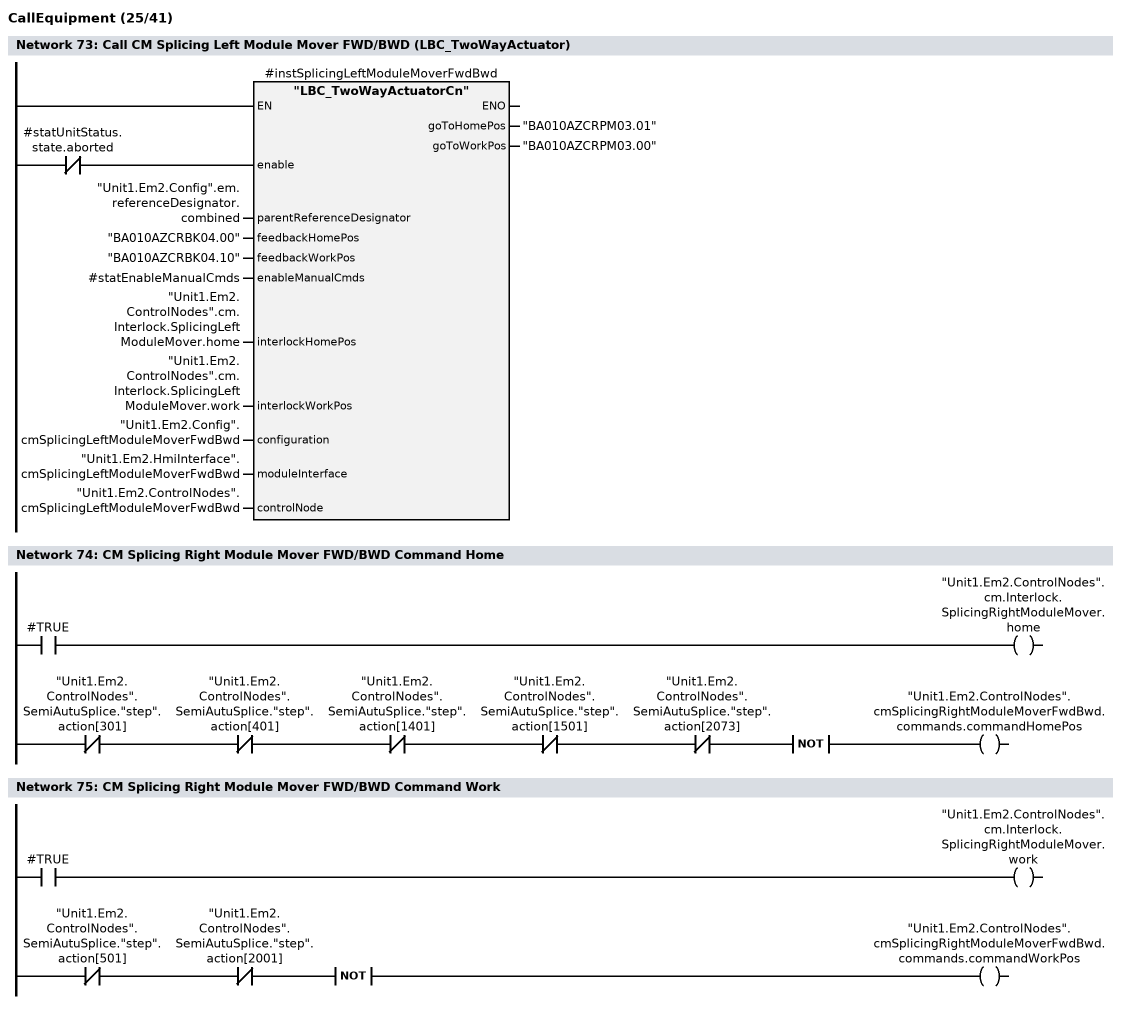
   RUNG wire#powerrail
      #instSplicingLeftModuleMoverFwdBwd(enable := wire#w1, parentReferenceDesignator := "Unit1.Em2.Config".em.referenceDesignator.combined, feedbackHomePos := "BA010AZCRBK04.00", feedbackWorkPos := "BA010AZCRBK04.10", enableManualCmds := #statEnableManualCmds, interlockHomePos := "Unit1.Em2.ControlNodes".cm.Interlock.SplicingLeftModuleMover.home, interlockWorkPos := "Unit1.Em2.ControlNodes".cm.Interlock.SplicingLeftModuleMover.work, configuration := "Unit1.Em2.Config".cmSplicingLeftModuleMoverFwdBwd, moduleInterface := "Unit1.Em2.HmiInterface".cmSplicingLeftModuleMoverFwdBwd, controlNode := "Unit1.Em2.ControlNodes".cmSplicingLeftModuleMoverFwdBwd, goToHomePos => "BA010AZCRPM03.01", goToWorkPos => "BA010AZCRPM03.00")
   END_RUNG
   RUNG wire#powerrail
      I_Contact( #statUnitStatus.state.aborted )
   END_RUNG wire#w1
   // the same network as SCL:
   #instSplicingLeftModuleMoverFwdBwd(enable := NOT #statUnitStatus.state.aborted,   // "LBC_TwoWayActuatorCn"
                           parentReferenceDesignator := "Unit1.Em2.Config".em.referenceDesignator.combined,
                           feedbackHomePos := "BA010AZCRBK04.00",
                           feedbackWorkPos := "BA010AZCRBK04.10",
                           enableManualCmds := #statEnableManualCmds,
                           interlockHomePos := "Unit1.Em2.ControlNodes".cm.Interlock.SplicingLeftModuleMover.home,
                           interlockWorkPos := "Unit1.Em2.ControlNodes".cm.Interlock.SplicingLeftModuleMover.work,
                           configuration := "Unit1.Em2.Config".cmSplicingLeftModuleMoverFwdBwd,
                           moduleInterface := "Unit1.Em2.HmiInterface".cmSplicingLeftModuleMoverFwdBwd,
                           controlNode := "Unit1.Em2.ControlNodes".cmSplicingLeftModuleMoverFwdBwd,
                           goToHomePos => "BA010AZCRPM03.01",
                           goToWorkPos => "BA010AZCRPM03.00");
END_REGION

REGION Network 74: CM Splicing Right Module Mover FWD/BWD Command Home
   RUNG wire#powerrail
      Contact( #TRUE )
      Coil( "Unit1.Em2.ControlNodes".cm.Interlock.SplicingRightModuleMover.home )
   END_RUNG
   RUNG wire#powerrail
      I_Contact( "Unit1.Em2.ControlNodes".SemiAutuSplice."step".action[301] )
      I_Contact( "Unit1.Em2.ControlNodes".SemiAutuSplice."step".action[401] )
      I_Contact( "Unit1.Em2.ControlNodes".SemiAutuSplice."step".action[1401] )
      I_Contact( "Unit1.Em2.ControlNodes".SemiAutuSplice."step".action[1501] )
      I_Contact( "Unit1.Em2.ControlNodes".SemiAutuSplice."step".action[2073] )
      Not()
      Coil( "Unit1.Em2.ControlNodes".cmSplicingRightModuleMoverFwdBwd.commands.commandHomePos )
   END_RUNG
   // the same network as SCL:
   "Unit1.Em2.ControlNodes".cm.Interlock.SplicingRightModuleMover.home := #TRUE;
   "Unit1.Em2.ControlNodes".cmSplicingRightModuleMoverFwdBwd.commands.commandHomePos := NOT (NOT "Unit1.Em2.ControlNodes".SemiAutuSplice."step".action[301] AND NOT "Unit1.Em2.ControlNodes".SemiAutuSplice."step".action[401] AND NOT "Unit1.Em2.ControlNodes".SemiAutuSplice."step".action[1401] AND NOT "Unit1.Em2.ControlNodes".SemiAutuSplice."step".action[1501] AND NOT "Unit1.Em2.ControlNodes".SemiAutuSplice."step".action[2073]);
END_REGION

REGION Network 75: CM Splicing Right Module Mover FWD/BWD Command Work
   RUNG wire#powerrail
      Contact( #TRUE )
      Coil( "Unit1.Em2.ControlNodes".cm.Interlock.SplicingRightModuleMover.work )
   END_RUNG
   RUNG wire#powerrail
      I_Contact( "Unit1.Em2.ControlNodes".SemiAutuSplice."step".action[501] )
      I_Contact( "Unit1.Em2.ControlNodes".SemiAutuSplice."step".action[2001] )
      Not()
      Coil( "Unit1.Em2.ControlNodes".cmSplicingRightModuleMoverFwdBwd.commands.commandWorkPos )
   END_RUNG
   // the same network as SCL:
   "Unit1.Em2.ControlNodes".cm.Interlock.SplicingRightModuleMover.work := #TRUE;
   "Unit1.Em2.ControlNodes".cmSplicingRightModuleMoverFwdBwd.commands.commandWorkPos := NOT (NOT "Unit1.Em2.ControlNodes".SemiAutuSplice."step".action[501] AND NOT "Unit1.Em2.ControlNodes".SemiAutuSplice."step".action[2001]);
END_REGION

REGION Network 76: Call CM Splicing Right Module Mover FWD/BWD (LBC_TwoWayActuator)
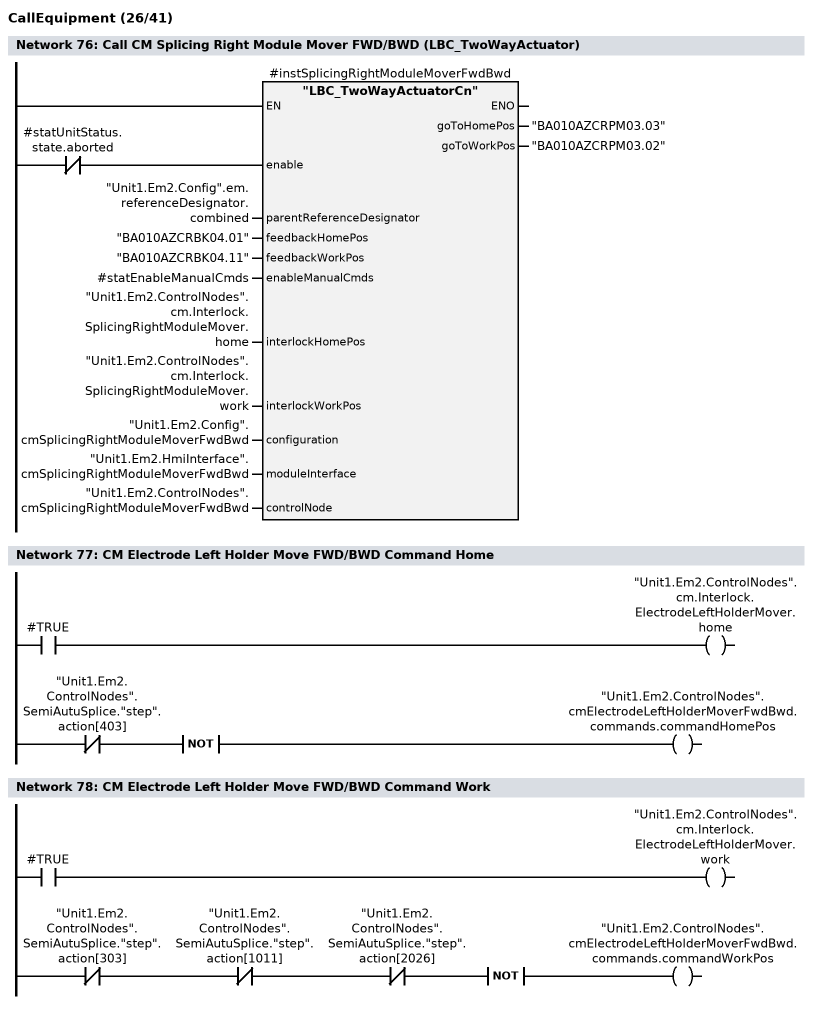
   RUNG wire#powerrail
      #instSplicingRightModuleMoverFwdBwd(enable := wire#w1, parentReferenceDesignator := "Unit1.Em2.Config".em.referenceDesignator.combined, feedbackHomePos := "BA010AZCRBK04.01", feedbackWorkPos := "BA010AZCRBK04.11", enableManualCmds := #statEnableManualCmds, interlockHomePos := "Unit1.Em2.ControlNodes".cm.Interlock.SplicingRightModuleMover.home, interlockWorkPos := "Unit1.Em2.ControlNodes".cm.Interlock.SplicingRightModuleMover.work, configuration := "Unit1.Em2.Config".cmSplicingRightModuleMoverFwdBwd, moduleInterface := "Unit1.Em2.HmiInterface".cmSplicingRightModuleMoverFwdBwd, controlNode := "Unit1.Em2.ControlNodes".cmSplicingRightModuleMoverFwdBwd, goToHomePos => "BA010AZCRPM03.03", goToWorkPos => "BA010AZCRPM03.02")
   END_RUNG
   RUNG wire#powerrail
      I_Contact( #statUnitStatus.state.aborted )
   END_RUNG wire#w1
   // the same network as SCL:
   #instSplicingRightModuleMoverFwdBwd(enable := NOT #statUnitStatus.state.aborted,   // "LBC_TwoWayActuatorCn"
                           parentReferenceDesignator := "Unit1.Em2.Config".em.referenceDesignator.combined,
                           feedbackHomePos := "BA010AZCRBK04.01",
                           feedbackWorkPos := "BA010AZCRBK04.11",
                           enableManualCmds := #statEnableManualCmds,
                           interlockHomePos := "Unit1.Em2.ControlNodes".cm.Interlock.SplicingRightModuleMover.home,
                           interlockWorkPos := "Unit1.Em2.ControlNodes".cm.Interlock.SplicingRightModuleMover.work,
                           configuration := "Unit1.Em2.Config".cmSplicingRightModuleMoverFwdBwd,
                           moduleInterface := "Unit1.Em2.HmiInterface".cmSplicingRightModuleMoverFwdBwd,
                           controlNode := "Unit1.Em2.ControlNodes".cmSplicingRightModuleMoverFwdBwd,
                           goToHomePos => "BA010AZCRPM03.03",
                           goToWorkPos => "BA010AZCRPM03.02");
END_REGION

REGION Network 77: CM Electrode Left Holder Move FWD/BWD Command Home
   RUNG wire#powerrail
      Contact( #TRUE )
      Coil( "Unit1.Em2.ControlNodes".cm.Interlock.ElectrodeLeftHolderMover.home )
   END_RUNG
   RUNG wire#powerrail
      I_Contact( "Unit1.Em2.ControlNodes".SemiAutuSplice."step".action[403] )
      Not()
      Coil( "Unit1.Em2.ControlNodes".cmElectrodeLeftHolderMoverFwdBwd.commands.commandHomePos )
   END_RUNG
   // the same network as SCL:
   "Unit1.Em2.ControlNodes".cm.Interlock.ElectrodeLeftHolderMover.home := #TRUE;
   "Unit1.Em2.ControlNodes".cmElectrodeLeftHolderMoverFwdBwd.commands.commandHomePos := NOT (NOT "Unit1.Em2.ControlNodes".SemiAutuSplice."step".action[403]);
END_REGION

REGION Network 78: CM Electrode Left Holder Move FWD/BWD Command Work
   RUNG wire#powerrail
      Contact( #TRUE )
      Coil( "Unit1.Em2.ControlNodes".cm.Interlock.ElectrodeLeftHolderMover.work )
   END_RUNG
   RUNG wire#powerrail
      I_Contact( "Unit1.Em2.ControlNodes".SemiAutuSplice."step".action[303] )
      I_Contact( "Unit1.Em2.ControlNodes".SemiAutuSplice."step".action[1011] )
      I_Contact( "Unit1.Em2.ControlNodes".SemiAutuSplice."step".action[2026] )
      Not()
      Coil( "Unit1.Em2.ControlNodes".cmElectrodeLeftHolderMoverFwdBwd.commands.commandWorkPos )
   END_RUNG
   // the same network as SCL:
   "Unit1.Em2.ControlNodes".cm.Interlock.ElectrodeLeftHolderMover.work := #TRUE;
   "Unit1.Em2.ControlNodes".cmElectrodeLeftHolderMoverFwdBwd.commands.commandWorkPos := NOT (NOT "Unit1.Em2.ControlNodes".SemiAutuSplice."step".action[303] AND NOT "Unit1.Em2.ControlNodes".SemiAutuSplice."step".action[1011] AND NOT "Unit1.Em2.ControlNodes".SemiAutuSplice."step".action[2026]);
END_REGION

REGION Network 79: Call CM Electrode Left Holder Move FWD/BWD (LBC_TwoWayActuator)
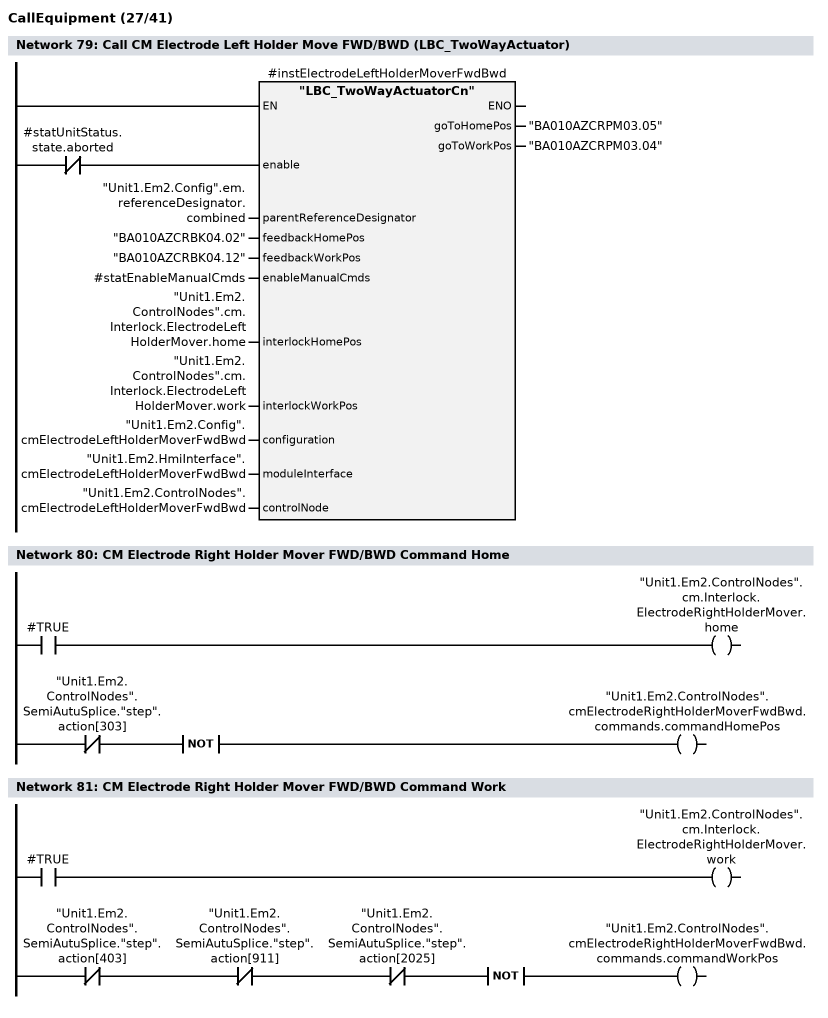
   RUNG wire#powerrail
      #instElectrodeLeftHolderMoverFwdBwd(enable := wire#w1, parentReferenceDesignator := "Unit1.Em2.Config".em.referenceDesignator.combined, feedbackHomePos := "BA010AZCRBK04.02", feedbackWorkPos := "BA010AZCRBK04.12", enableManualCmds := #statEnableManualCmds, interlockHomePos := "Unit1.Em2.ControlNodes".cm.Interlock.ElectrodeLeftHolderMover.home, interlockWorkPos := "Unit1.Em2.ControlNodes".cm.Interlock.ElectrodeLeftHolderMover.work, configuration := "Unit1.Em2.Config".cmElectrodeLeftHolderMoverFwdBwd, moduleInterface := "Unit1.Em2.HmiInterface".cmElectrodeLeftHolderMoverFwdBwd, controlNode := "Unit1.Em2.ControlNodes".cmElectrodeLeftHolderMoverFwdBwd, goToHomePos => "BA010AZCRPM03.05", goToWorkPos => "BA010AZCRPM03.04")
   END_RUNG
   RUNG wire#powerrail
      I_Contact( #statUnitStatus.state.aborted )
   END_RUNG wire#w1
   // the same network as SCL:
   #instElectrodeLeftHolderMoverFwdBwd(enable := NOT #statUnitStatus.state.aborted,   // "LBC_TwoWayActuatorCn"
                           parentReferenceDesignator := "Unit1.Em2.Config".em.referenceDesignator.combined,
                           feedbackHomePos := "BA010AZCRBK04.02",
                           feedbackWorkPos := "BA010AZCRBK04.12",
                           enableManualCmds := #statEnableManualCmds,
                           interlockHomePos := "Unit1.Em2.ControlNodes".cm.Interlock.ElectrodeLeftHolderMover.home,
                           interlockWorkPos := "Unit1.Em2.ControlNodes".cm.Interlock.ElectrodeLeftHolderMover.work,
                           configuration := "Unit1.Em2.Config".cmElectrodeLeftHolderMoverFwdBwd,
                           moduleInterface := "Unit1.Em2.HmiInterface".cmElectrodeLeftHolderMoverFwdBwd,
                           controlNode := "Unit1.Em2.ControlNodes".cmElectrodeLeftHolderMoverFwdBwd,
                           goToHomePos => "BA010AZCRPM03.05",
                           goToWorkPos => "BA010AZCRPM03.04");
END_REGION

REGION Network 80: CM Electrode Right Holder Mover FWD/BWD Command Home
   RUNG wire#powerrail
      Contact( #TRUE )
      Coil( "Unit1.Em2.ControlNodes".cm.Interlock.ElectrodeRightHolderMover.home )
   END_RUNG
   RUNG wire#powerrail
      I_Contact( "Unit1.Em2.ControlNodes".SemiAutuSplice."step".action[303] )
      Not()
      Coil( "Unit1.Em2.ControlNodes".cmElectrodeRightHolderMoverFwdBwd.commands.commandHomePos )
   END_RUNG
   // the same network as SCL:
   "Unit1.Em2.ControlNodes".cm.Interlock.ElectrodeRightHolderMover.home := #TRUE;
   "Unit1.Em2.ControlNodes".cmElectrodeRightHolderMoverFwdBwd.commands.commandHomePos := NOT (NOT "Unit1.Em2.ControlNodes".SemiAutuSplice."step".action[303]);
END_REGION

REGION Network 81: CM Electrode Right Holder Mover FWD/BWD Command Work
   RUNG wire#powerrail
      Contact( #TRUE )
      Coil( "Unit1.Em2.ControlNodes".cm.Interlock.ElectrodeRightHolderMover.work )
   END_RUNG
   RUNG wire#powerrail
      I_Contact( "Unit1.Em2.ControlNodes".SemiAutuSplice."step".action[403] )
      I_Contact( "Unit1.Em2.ControlNodes".SemiAutuSplice."step".action[911] )
      I_Contact( "Unit1.Em2.ControlNodes".SemiAutuSplice."step".action[2025] )
      Not()
      Coil( "Unit1.Em2.ControlNodes".cmElectrodeRightHolderMoverFwdBwd.commands.commandWorkPos )
   END_RUNG
   // the same network as SCL:
   "Unit1.Em2.ControlNodes".cm.Interlock.ElectrodeRightHolderMover.work := #TRUE;
   "Unit1.Em2.ControlNodes".cmElectrodeRightHolderMoverFwdBwd.commands.commandWorkPos := NOT (NOT "Unit1.Em2.ControlNodes".SemiAutuSplice."step".action[403] AND NOT "Unit1.Em2.ControlNodes".SemiAutuSplice."step".action[911] AND NOT "Unit1.Em2.ControlNodes".SemiAutuSplice."step".action[2025]);
END_REGION

REGION Network 82: Call CM Electrode Right Holder Mover FWD/BWD (LBC_TwoWayActuator)
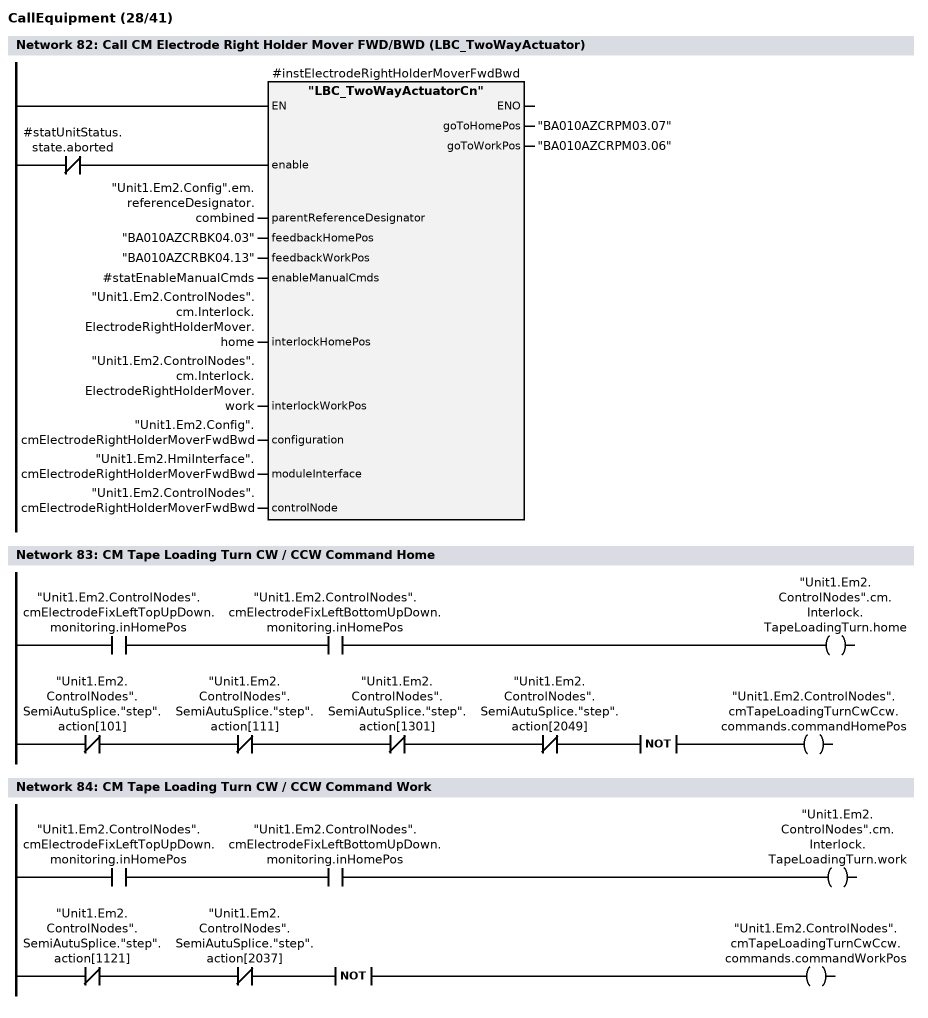
   RUNG wire#powerrail
      #instElectrodeRightHolderMoverFwdBwd(enable := wire#w1, parentReferenceDesignator := "Unit1.Em2.Config".em.referenceDesignator.combined, feedbackHomePos := "BA010AZCRBK04.03", feedbackWorkPos := "BA010AZCRBK04.13", enableManualCmds := #statEnableManualCmds, interlockHomePos := "Unit1.Em2.ControlNodes".cm.Interlock.ElectrodeRightHolderMover.home, interlockWorkPos := "Unit1.Em2.ControlNodes".cm.Interlock.ElectrodeRightHolderMover.work, configuration := "Unit1.Em2.Config".cmElectrodeRightHolderMoverFwdBwd, moduleInterface := "Unit1.Em2.HmiInterface".cmElectrodeRightHolderMoverFwdBwd, controlNode := "Unit1.Em2.ControlNodes".cmElectrodeRightHolderMoverFwdBwd, goToHomePos => "BA010AZCRPM03.07", goToWorkPos => "BA010AZCRPM03.06")
   END_RUNG
   RUNG wire#powerrail
      I_Contact( #statUnitStatus.state.aborted )
   END_RUNG wire#w1
   // the same network as SCL:
   #instElectrodeRightHolderMoverFwdBwd(enable := NOT #statUnitStatus.state.aborted,   // "LBC_TwoWayActuatorCn"
                           parentReferenceDesignator := "Unit1.Em2.Config".em.referenceDesignator.combined,
                           feedbackHomePos := "BA010AZCRBK04.03",
                           feedbackWorkPos := "BA010AZCRBK04.13",
                           enableManualCmds := #statEnableManualCmds,
                           interlockHomePos := "Unit1.Em2.ControlNodes".cm.Interlock.ElectrodeRightHolderMover.home,
                           interlockWorkPos := "Unit1.Em2.ControlNodes".cm.Interlock.ElectrodeRightHolderMover.work,
                           configuration := "Unit1.Em2.Config".cmElectrodeRightHolderMoverFwdBwd,
                           moduleInterface := "Unit1.Em2.HmiInterface".cmElectrodeRightHolderMoverFwdBwd,
                           controlNode := "Unit1.Em2.ControlNodes".cmElectrodeRightHolderMoverFwdBwd,
                           goToHomePos => "BA010AZCRPM03.07",
                           goToWorkPos => "BA010AZCRPM03.06");
END_REGION

REGION Network 83: CM Tape Loading Turn CW / CCW Command Home
   RUNG wire#powerrail
      Contact( "Unit1.Em2.ControlNodes".cmElectrodeFixLeftTopUpDown.monitoring.inHomePos )
      Contact( "Unit1.Em2.ControlNodes".cmElectrodeFixLeftBottomUpDown.monitoring.inHomePos )
      Coil( "Unit1.Em2.ControlNodes".cm.Interlock.TapeLoadingTurn.home )
   END_RUNG
   RUNG wire#powerrail
      I_Contact( "Unit1.Em2.ControlNodes".SemiAutuSplice."step".action[101] )
      I_Contact( "Unit1.Em2.ControlNodes".SemiAutuSplice."step".action[111] )
      I_Contact( "Unit1.Em2.ControlNodes".SemiAutuSplice."step".action[1301] )
      I_Contact( "Unit1.Em2.ControlNodes".SemiAutuSplice."step".action[2049] )
      Not()
      Coil( "Unit1.Em2.ControlNodes".cmTapeLoadingTurnCwCcw.commands.commandHomePos )
   END_RUNG
   // the same network as SCL:
   "Unit1.Em2.ControlNodes".cm.Interlock.TapeLoadingTurn.home := "Unit1.Em2.ControlNodes".cmElectrodeFixLeftTopUpDown.monitoring.inHomePos AND "Unit1.Em2.ControlNodes".cmElectrodeFixLeftBottomUpDown.monitoring.inHomePos;
   "Unit1.Em2.ControlNodes".cmTapeLoadingTurnCwCcw.commands.commandHomePos := NOT (NOT "Unit1.Em2.ControlNodes".SemiAutuSplice."step".action[101] AND NOT "Unit1.Em2.ControlNodes".SemiAutuSplice."step".action[111] AND NOT "Unit1.Em2.ControlNodes".SemiAutuSplice."step".action[1301] AND NOT "Unit1.Em2.ControlNodes".SemiAutuSplice."step".action[2049]);
END_REGION

REGION Network 84: CM Tape Loading Turn CW / CCW Command Work
   RUNG wire#powerrail
      Contact( "Unit1.Em2.ControlNodes".cmElectrodeFixLeftTopUpDown.monitoring.inHomePos )
      Contact( "Unit1.Em2.ControlNodes".cmElectrodeFixLeftBottomUpDown.monitoring.inHomePos )
      Coil( "Unit1.Em2.ControlNodes".cm.Interlock.TapeLoadingTurn.work )
   END_RUNG
   RUNG wire#powerrail
      I_Contact( "Unit1.Em2.ControlNodes".SemiAutuSplice."step".action[1121] )
      I_Contact( "Unit1.Em2.ControlNodes".SemiAutuSplice."step".action[2037] )
      Not()
      Coil( "Unit1.Em2.ControlNodes".cmTapeLoadingTurnCwCcw.commands.commandWorkPos )
   END_RUNG
   // the same network as SCL:
   "Unit1.Em2.ControlNodes".cm.Interlock.TapeLoadingTurn.work := "Unit1.Em2.ControlNodes".cmElectrodeFixLeftTopUpDown.monitoring.inHomePos AND "Unit1.Em2.ControlNodes".cmElectrodeFixLeftBottomUpDown.monitoring.inHomePos;
   "Unit1.Em2.ControlNodes".cmTapeLoadingTurnCwCcw.commands.commandWorkPos := NOT (NOT "Unit1.Em2.ControlNodes".SemiAutuSplice."step".action[1121] AND NOT "Unit1.Em2.ControlNodes".SemiAutuSplice."step".action[2037]);
END_REGION

REGION Network 85: Call CM Tape Loading Turn CW / CCW (LBC_TwoWayActuator)
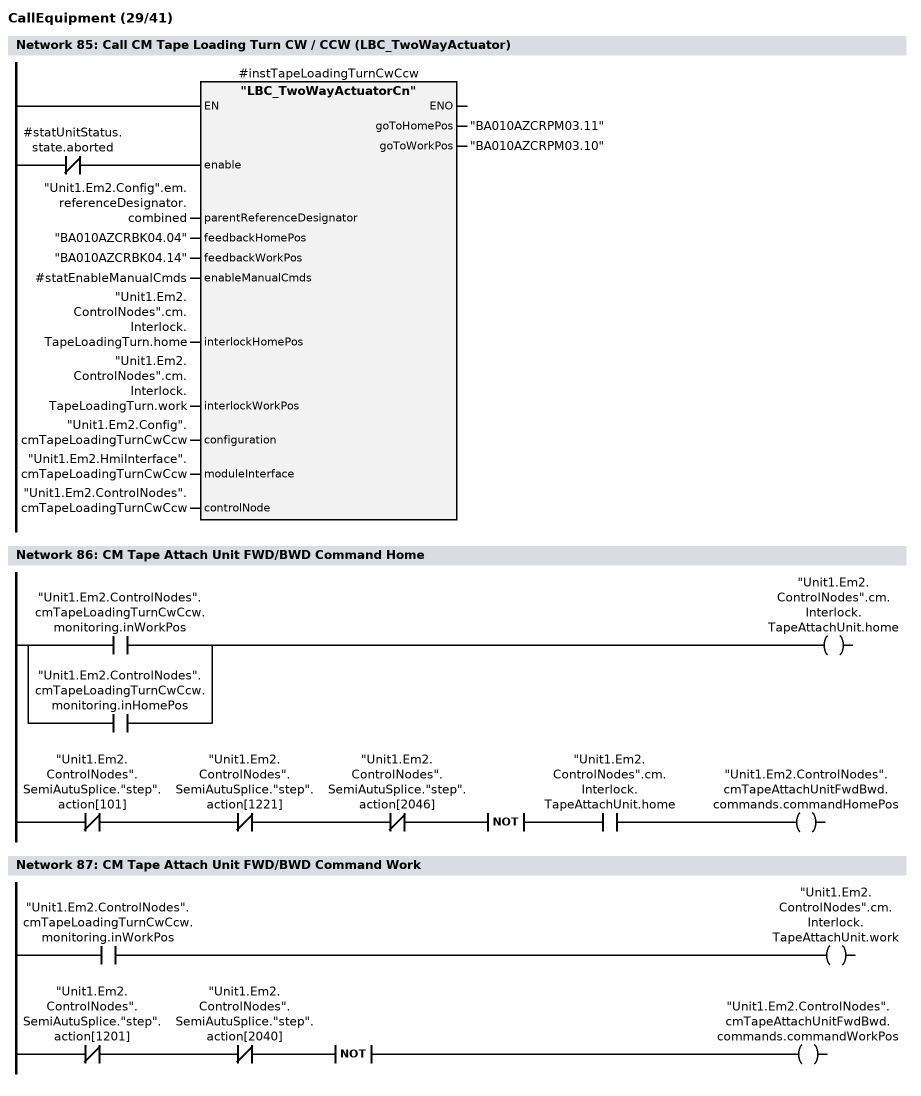
   RUNG wire#powerrail
      #instTapeLoadingTurnCwCcw(enable := wire#w1, parentReferenceDesignator := "Unit1.Em2.Config".em.referenceDesignator.combined, feedbackHomePos := "BA010AZCRBK04.04", feedbackWorkPos := "BA010AZCRBK04.14", enableManualCmds := #statEnableManualCmds, interlockHomePos := "Unit1.Em2.ControlNodes".cm.Interlock.TapeLoadingTurn.home, interlockWorkPos := "Unit1.Em2.ControlNodes".cm.Interlock.TapeLoadingTurn.work, configuration := "Unit1.Em2.Config".cmTapeLoadingTurnCwCcw, moduleInterface := "Unit1.Em2.HmiInterface".cmTapeLoadingTurnCwCcw, controlNode := "Unit1.Em2.ControlNodes".cmTapeLoadingTurnCwCcw, goToHomePos => "BA010AZCRPM03.11", goToWorkPos => "BA010AZCRPM03.10")
   END_RUNG
   RUNG wire#powerrail
      I_Contact( #statUnitStatus.state.aborted )
   END_RUNG wire#w1
   // the same network as SCL:
   #instTapeLoadingTurnCwCcw(enable := NOT #statUnitStatus.state.aborted,   // "LBC_TwoWayActuatorCn"
                           parentReferenceDesignator := "Unit1.Em2.Config".em.referenceDesignator.combined,
                           feedbackHomePos := "BA010AZCRBK04.04",
                           feedbackWorkPos := "BA010AZCRBK04.14",
                           enableManualCmds := #statEnableManualCmds,
                           interlockHomePos := "Unit1.Em2.ControlNodes".cm.Interlock.TapeLoadingTurn.home,
                           interlockWorkPos := "Unit1.Em2.ControlNodes".cm.Interlock.TapeLoadingTurn.work,
                           configuration := "Unit1.Em2.Config".cmTapeLoadingTurnCwCcw,
                           moduleInterface := "Unit1.Em2.HmiInterface".cmTapeLoadingTurnCwCcw,
                           controlNode := "Unit1.Em2.ControlNodes".cmTapeLoadingTurnCwCcw,
                           goToHomePos => "BA010AZCRPM03.11",
                           goToWorkPos => "BA010AZCRPM03.10");
END_REGION

REGION Network 86: CM Tape Attach Unit FWD/BWD Command Home
   RUNG wire#powerrail
      Contact( "Unit1.Em2.ControlNodes".cmTapeLoadingTurnCwCcw.monitoring.inWorkPos )
      wire#w1
      Coil( "Unit1.Em2.ControlNodes".cm.Interlock.TapeAttachUnit.home )
   END_RUNG
   RUNG wire#powerrail
      Contact( "Unit1.Em2.ControlNodes".cmTapeLoadingTurnCwCcw.monitoring.inHomePos )
   END_RUNG wire#w1
   RUNG wire#powerrail
      I_Contact( "Unit1.Em2.ControlNodes".SemiAutuSplice."step".action[101] )
      I_Contact( "Unit1.Em2.ControlNodes".SemiAutuSplice."step".action[1221] )
      I_Contact( "Unit1.Em2.ControlNodes".SemiAutuSplice."step".action[2046] )
      Not()
      Contact( "Unit1.Em2.ControlNodes".cm.Interlock.TapeAttachUnit.home )
      Coil( "Unit1.Em2.ControlNodes".cmTapeAttachUnitFwdBwd.commands.commandHomePos )
   END_RUNG
   // the same network as SCL:
   "Unit1.Em2.ControlNodes".cm.Interlock.TapeAttachUnit.home := "Unit1.Em2.ControlNodes".cmTapeLoadingTurnCwCcw.monitoring.inWorkPos OR "Unit1.Em2.ControlNodes".cmTapeLoadingTurnCwCcw.monitoring.inHomePos;
   "Unit1.Em2.ControlNodes".cmTapeAttachUnitFwdBwd.commands.commandHomePos := NOT (NOT "Unit1.Em2.ControlNodes".SemiAutuSplice."step".action[101] AND NOT "Unit1.Em2.ControlNodes".SemiAutuSplice."step".action[1221] AND NOT "Unit1.Em2.ControlNodes".SemiAutuSplice."step".action[2046]) AND "Unit1.Em2.ControlNodes".cm.Interlock.TapeAttachUnit.home;
END_REGION

REGION Network 87: CM Tape Attach Unit FWD/BWD Command Work
   RUNG wire#powerrail
      Contact( "Unit1.Em2.ControlNodes".cmTapeLoadingTurnCwCcw.monitoring.inWorkPos )
      Coil( "Unit1.Em2.ControlNodes".cm.Interlock.TapeAttachUnit.work )
   END_RUNG
   RUNG wire#powerrail
      I_Contact( "Unit1.Em2.ControlNodes".SemiAutuSplice."step".action[1201] )
      I_Contact( "Unit1.Em2.ControlNodes".SemiAutuSplice."step".action[2040] )
      Not()
      Coil( "Unit1.Em2.ControlNodes".cmTapeAttachUnitFwdBwd.commands.commandWorkPos )
   END_RUNG
   // the same network as SCL:
   "Unit1.Em2.ControlNodes".cm.Interlock.TapeAttachUnit.work := "Unit1.Em2.ControlNodes".cmTapeLoadingTurnCwCcw.monitoring.inWorkPos;
   "Unit1.Em2.ControlNodes".cmTapeAttachUnitFwdBwd.commands.commandWorkPos := NOT (NOT "Unit1.Em2.ControlNodes".SemiAutuSplice."step".action[1201] AND NOT "Unit1.Em2.ControlNodes".SemiAutuSplice."step".action[2040]);
END_REGION

REGION Network 88: Call CM Tape Attach Unit FWD/BWD (LBC_TwoWayActuator)
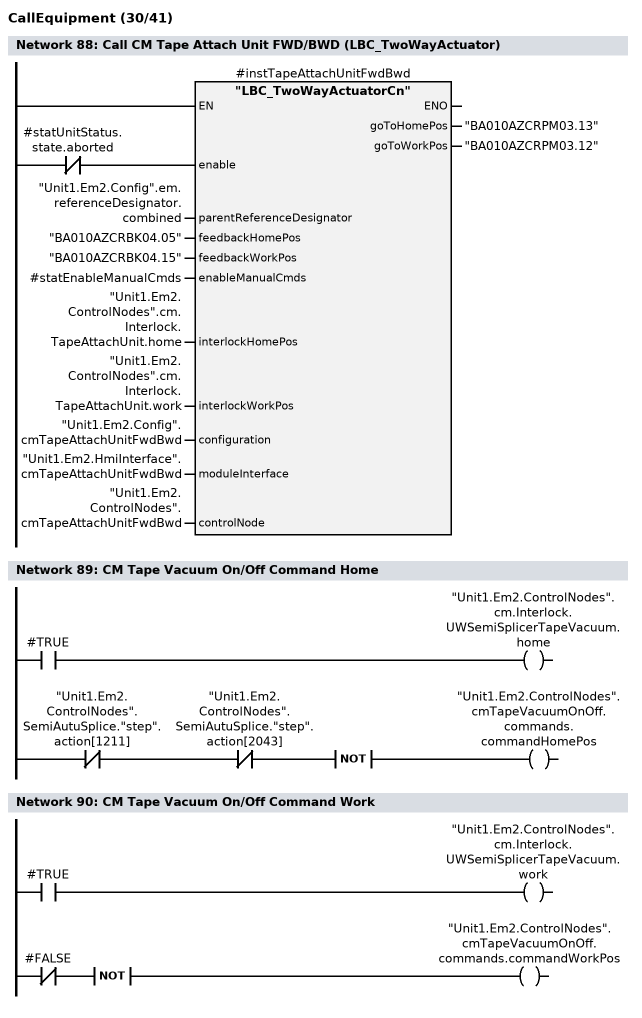
   RUNG wire#powerrail
      #instTapeAttachUnitFwdBwd(enable := wire#w1, parentReferenceDesignator := "Unit1.Em2.Config".em.referenceDesignator.combined, feedbackHomePos := "BA010AZCRBK04.05", feedbackWorkPos := "BA010AZCRBK04.15", enableManualCmds := #statEnableManualCmds, interlockHomePos := "Unit1.Em2.ControlNodes".cm.Interlock.TapeAttachUnit.home, interlockWorkPos := "Unit1.Em2.ControlNodes".cm.Interlock.TapeAttachUnit.work, configuration := "Unit1.Em2.Config".cmTapeAttachUnitFwdBwd, moduleInterface := "Unit1.Em2.HmiInterface".cmTapeAttachUnitFwdBwd, controlNode := "Unit1.Em2.ControlNodes".cmTapeAttachUnitFwdBwd, goToHomePos => "BA010AZCRPM03.13", goToWorkPos => "BA010AZCRPM03.12")
   END_RUNG
   RUNG wire#powerrail
      I_Contact( #statUnitStatus.state.aborted )
   END_RUNG wire#w1
   // the same network as SCL:
   #instTapeAttachUnitFwdBwd(enable := NOT #statUnitStatus.state.aborted,   // "LBC_TwoWayActuatorCn"
                           parentReferenceDesignator := "Unit1.Em2.Config".em.referenceDesignator.combined,
                           feedbackHomePos := "BA010AZCRBK04.05",
                           feedbackWorkPos := "BA010AZCRBK04.15",
                           enableManualCmds := #statEnableManualCmds,
                           interlockHomePos := "Unit1.Em2.ControlNodes".cm.Interlock.TapeAttachUnit.home,
                           interlockWorkPos := "Unit1.Em2.ControlNodes".cm.Interlock.TapeAttachUnit.work,
                           configuration := "Unit1.Em2.Config".cmTapeAttachUnitFwdBwd,
                           moduleInterface := "Unit1.Em2.HmiInterface".cmTapeAttachUnitFwdBwd,
                           controlNode := "Unit1.Em2.ControlNodes".cmTapeAttachUnitFwdBwd,
                           goToHomePos => "BA010AZCRPM03.13",
                           goToWorkPos => "BA010AZCRPM03.12");
END_REGION

REGION Network 89: CM Tape Vacuum On/Off Command Home
   RUNG wire#powerrail
      Contact( #TRUE )
      Coil( "Unit1.Em2.ControlNodes".cm.Interlock.UWSemiSplicerTapeVacuum.home )
   END_RUNG
   RUNG wire#powerrail
      I_Contact( "Unit1.Em2.ControlNodes".SemiAutuSplice."step".action[1211] )
      I_Contact( "Unit1.Em2.ControlNodes".SemiAutuSplice."step".action[2043] )
      Not()
      Coil( "Unit1.Em2.ControlNodes".cmTapeVacuumOnOff.commands.commandHomePos )
   END_RUNG
   // the same network as SCL:
   "Unit1.Em2.ControlNodes".cm.Interlock.UWSemiSplicerTapeVacuum.home := #TRUE;
   "Unit1.Em2.ControlNodes".cmTapeVacuumOnOff.commands.commandHomePos := NOT (NOT "Unit1.Em2.ControlNodes".SemiAutuSplice."step".action[1211] AND NOT "Unit1.Em2.ControlNodes".SemiAutuSplice."step".action[2043]);
END_REGION

REGION Network 90: CM Tape Vacuum On/Off Command Work
   RUNG wire#powerrail
      Contact( #TRUE )
      Coil( "Unit1.Em2.ControlNodes".cm.Interlock.UWSemiSplicerTapeVacuum.work )
   END_RUNG
   RUNG wire#powerrail
      I_Contact( #FALSE )
      Not()
      Coil( "Unit1.Em2.ControlNodes".cmTapeVacuumOnOff.commands.commandWorkPos )
   END_RUNG
   // the same network as SCL:
   "Unit1.Em2.ControlNodes".cm.Interlock.UWSemiSplicerTapeVacuum.work := #TRUE;
   "Unit1.Em2.ControlNodes".cmTapeVacuumOnOff.commands.commandWorkPos := NOT (NOT #FALSE);
END_REGION

REGION Network 91: Call CM Tape Vacuum On/Off (LBC_TwoWayActuator)
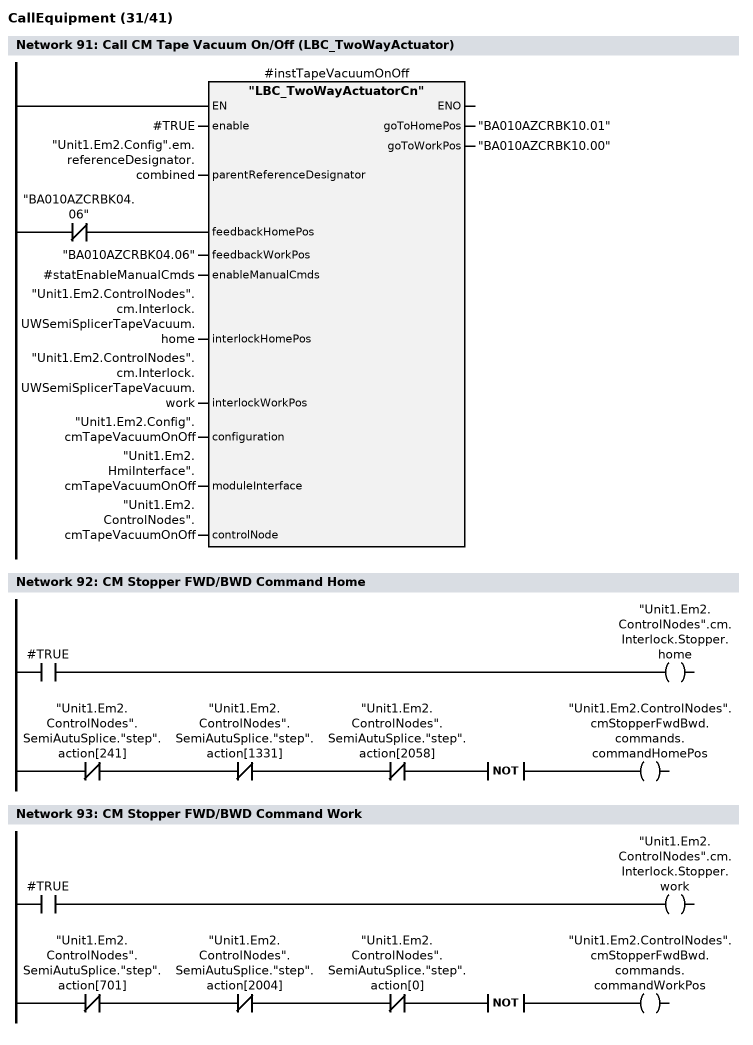
   RUNG wire#powerrail
      #instTapeVacuumOnOff(feedbackHomePos := wire#w1, enable := #TRUE, parentReferenceDesignator := "Unit1.Em2.Config".em.referenceDesignator.combined, feedbackWorkPos := "BA010AZCRBK04.06", enableManualCmds := #statEnableManualCmds, interlockHomePos := "Unit1.Em2.ControlNodes".cm.Interlock.UWSemiSplicerTapeVacuum.home, interlockWorkPos := "Unit1.Em2.ControlNodes".cm.Interlock.UWSemiSplicerTapeVacuum.work, configuration := "Unit1.Em2.Config".cmTapeVacuumOnOff, moduleInterface := "Unit1.Em2.HmiInterface".cmTapeVacuumOnOff, controlNode := "Unit1.Em2.ControlNodes".cmTapeVacuumOnOff, goToHomePos => "BA010AZCRBK10.01", goToWorkPos => "BA010AZCRBK10.00")
   END_RUNG
   RUNG wire#powerrail
      I_Contact( "BA010AZCRBK04.06" )
   END_RUNG wire#w1
   // the same network as SCL:
   #instTapeVacuumOnOff(enable := #TRUE,   // "LBC_TwoWayActuatorCn"
                        parentReferenceDesignator := "Unit1.Em2.Config".em.referenceDesignator.combined,
                        feedbackHomePos := NOT "BA010AZCRBK04.06",
                        feedbackWorkPos := "BA010AZCRBK04.06",
                        enableManualCmds := #statEnableManualCmds,
                        interlockHomePos := "Unit1.Em2.ControlNodes".cm.Interlock.UWSemiSplicerTapeVacuum.home,
                        interlockWorkPos := "Unit1.Em2.ControlNodes".cm.Interlock.UWSemiSplicerTapeVacuum.work,
                        configuration := "Unit1.Em2.Config".cmTapeVacuumOnOff,
                        moduleInterface := "Unit1.Em2.HmiInterface".cmTapeVacuumOnOff,
                        controlNode := "Unit1.Em2.ControlNodes".cmTapeVacuumOnOff,
                        goToHomePos => "BA010AZCRBK10.01",
                        goToWorkPos => "BA010AZCRBK10.00");
END_REGION

REGION Network 92: CM Stopper FWD/BWD Command Home
   RUNG wire#powerrail
      Contact( #TRUE )
      Coil( "Unit1.Em2.ControlNodes".cm.Interlock.Stopper.home )
   END_RUNG
   RUNG wire#powerrail
      I_Contact( "Unit1.Em2.ControlNodes".SemiAutuSplice."step".action[241] )
      I_Contact( "Unit1.Em2.ControlNodes".SemiAutuSplice."step".action[1331] )
      I_Contact( "Unit1.Em2.ControlNodes".SemiAutuSplice."step".action[2058] )
      Not()
      Coil( "Unit1.Em2.ControlNodes".cmStopperFwdBwd.commands.commandHomePos )
   END_RUNG
   // the same network as SCL:
   "Unit1.Em2.ControlNodes".cm.Interlock.Stopper.home := #TRUE;
   "Unit1.Em2.ControlNodes".cmStopperFwdBwd.commands.commandHomePos := NOT (NOT "Unit1.Em2.ControlNodes".SemiAutuSplice."step".action[241] AND NOT "Unit1.Em2.ControlNodes".SemiAutuSplice."step".action[1331] AND NOT "Unit1.Em2.ControlNodes".SemiAutuSplice."step".action[2058]);
END_REGION

REGION Network 93: CM Stopper FWD/BWD Command Work
   RUNG wire#powerrail
      Contact( #TRUE )
      Coil( "Unit1.Em2.ControlNodes".cm.Interlock.Stopper.work )
   END_RUNG
   RUNG wire#powerrail
      I_Contact( "Unit1.Em2.ControlNodes".SemiAutuSplice."step".action[701] )
      I_Contact( "Unit1.Em2.ControlNodes".SemiAutuSplice."step".action[2004] )
      I_Contact( "Unit1.Em2.ControlNodes".SemiAutuSplice."step".action[0] )
      Not()
      Coil( "Unit1.Em2.ControlNodes".cmStopperFwdBwd.commands.commandWorkPos )
   END_RUNG
   // the same network as SCL:
   "Unit1.Em2.ControlNodes".cm.Interlock.Stopper.work := #TRUE;
   "Unit1.Em2.ControlNodes".cmStopperFwdBwd.commands.commandWorkPos := NOT (NOT "Unit1.Em2.ControlNodes".SemiAutuSplice."step".action[701] AND NOT "Unit1.Em2.ControlNodes".SemiAutuSplice."step".action[2004] AND NOT "Unit1.Em2.ControlNodes".SemiAutuSplice."step".action[0]);
END_REGION

REGION Network 94: Call CM Stopper FWD/BWD (LBC_TwoWayActuator)
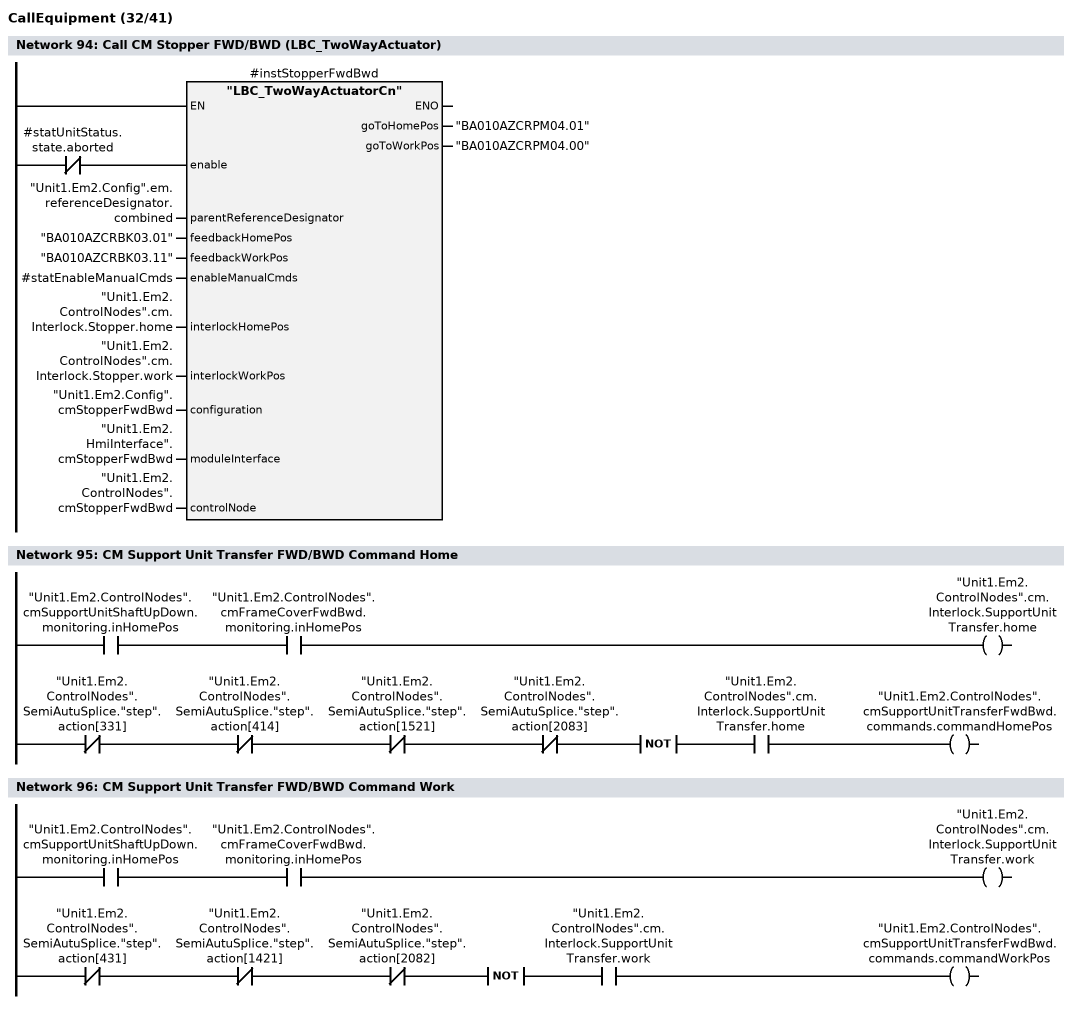
   RUNG wire#powerrail
      #instStopperFwdBwd(enable := wire#w1, parentReferenceDesignator := "Unit1.Em2.Config".em.referenceDesignator.combined, feedbackHomePos := "BA010AZCRBK03.01", feedbackWorkPos := "BA010AZCRBK03.11", enableManualCmds := #statEnableManualCmds, interlockHomePos := "Unit1.Em2.ControlNodes".cm.Interlock.Stopper.home, interlockWorkPos := "Unit1.Em2.ControlNodes".cm.Interlock.Stopper.work, configuration := "Unit1.Em2.Config".cmStopperFwdBwd, moduleInterface := "Unit1.Em2.HmiInterface".cmStopperFwdBwd, controlNode := "Unit1.Em2.ControlNodes".cmStopperFwdBwd, goToHomePos => "BA010AZCRPM04.01", goToWorkPos => "BA010AZCRPM04.00")
   END_RUNG
   RUNG wire#powerrail
      I_Contact( #statUnitStatus.state.aborted )
   END_RUNG wire#w1
   // the same network as SCL:
   #instStopperFwdBwd(enable := NOT #statUnitStatus.state.aborted,   // "LBC_TwoWayActuatorCn"
                      parentReferenceDesignator := "Unit1.Em2.Config".em.referenceDesignator.combined,
                      feedbackHomePos := "BA010AZCRBK03.01",
                      feedbackWorkPos := "BA010AZCRBK03.11",
                      enableManualCmds := #statEnableManualCmds,
                      interlockHomePos := "Unit1.Em2.ControlNodes".cm.Interlock.Stopper.home,
                      interlockWorkPos := "Unit1.Em2.ControlNodes".cm.Interlock.Stopper.work,
                      configuration := "Unit1.Em2.Config".cmStopperFwdBwd,
                      moduleInterface := "Unit1.Em2.HmiInterface".cmStopperFwdBwd,
                      controlNode := "Unit1.Em2.ControlNodes".cmStopperFwdBwd,
                      goToHomePos => "BA010AZCRPM04.01",
                      goToWorkPos => "BA010AZCRPM04.00");
END_REGION

REGION Network 95: CM Support Unit Transfer FWD/BWD Command Home
   RUNG wire#powerrail
      Contact( "Unit1.Em2.ControlNodes".cmSupportUnitShaftUpDown.monitoring.inHomePos )
      Contact( "Unit1.Em2.ControlNodes".cmFrameCoverFwdBwd.monitoring.inHomePos )
      Coil( "Unit1.Em2.ControlNodes".cm.Interlock.SupportUnitTransfer.home )
   END_RUNG
   RUNG wire#powerrail
      I_Contact( "Unit1.Em2.ControlNodes".SemiAutuSplice."step".action[331] )
      I_Contact( "Unit1.Em2.ControlNodes".SemiAutuSplice."step".action[414] )
      I_Contact( "Unit1.Em2.ControlNodes".SemiAutuSplice."step".action[1521] )
      I_Contact( "Unit1.Em2.ControlNodes".SemiAutuSplice."step".action[2083] )
      Not()
      Contact( "Unit1.Em2.ControlNodes".cm.Interlock.SupportUnitTransfer.home )
      Coil( "Unit1.Em2.ControlNodes".cmSupportUnitTransferFwdBwd.commands.commandHomePos )
   END_RUNG
   // the same network as SCL:
   "Unit1.Em2.ControlNodes".cm.Interlock.SupportUnitTransfer.home := "Unit1.Em2.ControlNodes".cmSupportUnitShaftUpDown.monitoring.inHomePos AND "Unit1.Em2.ControlNodes".cmFrameCoverFwdBwd.monitoring.inHomePos;
   "Unit1.Em2.ControlNodes".cmSupportUnitTransferFwdBwd.commands.commandHomePos := NOT (NOT "Unit1.Em2.ControlNodes".SemiAutuSplice."step".action[331] AND NOT "Unit1.Em2.ControlNodes".SemiAutuSplice."step".action[414] AND NOT "Unit1.Em2.ControlNodes".SemiAutuSplice."step".action[1521] AND NOT "Unit1.Em2.ControlNodes".SemiAutuSplice."step".action[2083]) AND "Unit1.Em2.ControlNodes".cm.Interlock.SupportUnitTransfer.home;
END_REGION

REGION Network 96: CM Support Unit Transfer FWD/BWD Command Work
   RUNG wire#powerrail
      Contact( "Unit1.Em2.ControlNodes".cmSupportUnitShaftUpDown.monitoring.inHomePos )
      Contact( "Unit1.Em2.ControlNodes".cmFrameCoverFwdBwd.monitoring.inHomePos )
      Coil( "Unit1.Em2.ControlNodes".cm.Interlock.SupportUnitTransfer.work )
   END_RUNG
   RUNG wire#powerrail
      I_Contact( "Unit1.Em2.ControlNodes".SemiAutuSplice."step".action[431] )
      I_Contact( "Unit1.Em2.ControlNodes".SemiAutuSplice."step".action[1421] )
      I_Contact( "Unit1.Em2.ControlNodes".SemiAutuSplice."step".action[2082] )
      Not()
      Contact( "Unit1.Em2.ControlNodes".cm.Interlock.SupportUnitTransfer.work )
      Coil( "Unit1.Em2.ControlNodes".cmSupportUnitTransferFwdBwd.commands.commandWorkPos )
   END_RUNG
   // the same network as SCL:
   "Unit1.Em2.ControlNodes".cm.Interlock.SupportUnitTransfer.work := "Unit1.Em2.ControlNodes".cmSupportUnitShaftUpDown.monitoring.inHomePos AND "Unit1.Em2.ControlNodes".cmFrameCoverFwdBwd.monitoring.inHomePos;
   "Unit1.Em2.ControlNodes".cmSupportUnitTransferFwdBwd.commands.commandWorkPos := NOT (NOT "Unit1.Em2.ControlNodes".SemiAutuSplice."step".action[431] AND NOT "Unit1.Em2.ControlNodes".SemiAutuSplice."step".action[1421] AND NOT "Unit1.Em2.ControlNodes".SemiAutuSplice."step".action[2082]) AND "Unit1.Em2.ControlNodes".cm.Interlock.SupportUnitTransfer.work;
END_REGION

REGION Network 97: Call CM Support Unit Transfer FWD/BWD (LBC_TwoWayActuator)
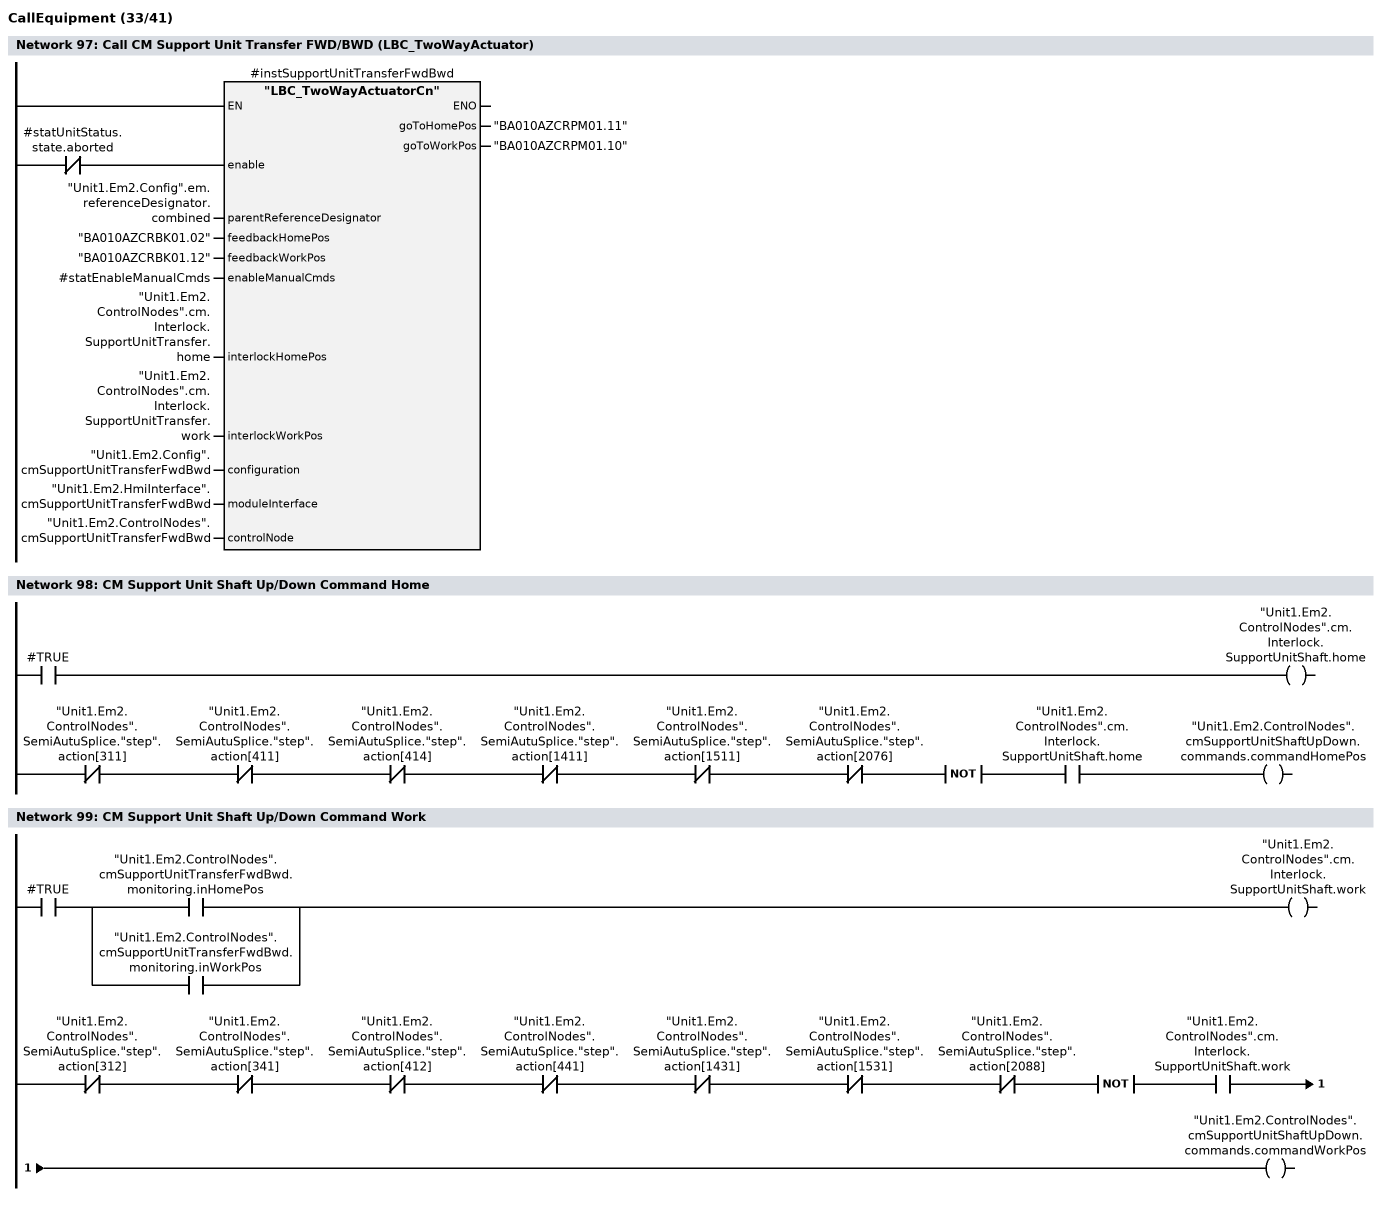
   RUNG wire#powerrail
      #instSupportUnitTransferFwdBwd(enable := wire#w1, parentReferenceDesignator := "Unit1.Em2.Config".em.referenceDesignator.combined, feedbackHomePos := "BA010AZCRBK01.02", feedbackWorkPos := "BA010AZCRBK01.12", enableManualCmds := #statEnableManualCmds, interlockHomePos := "Unit1.Em2.ControlNodes".cm.Interlock.SupportUnitTransfer.home, interlockWorkPos := "Unit1.Em2.ControlNodes".cm.Interlock.SupportUnitTransfer.work, configuration := "Unit1.Em2.Config".cmSupportUnitTransferFwdBwd, moduleInterface := "Unit1.Em2.HmiInterface".cmSupportUnitTransferFwdBwd, controlNode := "Unit1.Em2.ControlNodes".cmSupportUnitTransferFwdBwd, goToHomePos => "BA010AZCRPM01.11", goToWorkPos => "BA010AZCRPM01.10")
   END_RUNG
   RUNG wire#powerrail
      I_Contact( #statUnitStatus.state.aborted )
   END_RUNG wire#w1
   // the same network as SCL:
   #instSupportUnitTransferFwdBwd(enable := NOT #statUnitStatus.state.aborted,   // "LBC_TwoWayActuatorCn"
                           parentReferenceDesignator := "Unit1.Em2.Config".em.referenceDesignator.combined,
                           feedbackHomePos := "BA010AZCRBK01.02",
                           feedbackWorkPos := "BA010AZCRBK01.12",
                           enableManualCmds := #statEnableManualCmds,
                           interlockHomePos := "Unit1.Em2.ControlNodes".cm.Interlock.SupportUnitTransfer.home,
                           interlockWorkPos := "Unit1.Em2.ControlNodes".cm.Interlock.SupportUnitTransfer.work,
                           configuration := "Unit1.Em2.Config".cmSupportUnitTransferFwdBwd,
                           moduleInterface := "Unit1.Em2.HmiInterface".cmSupportUnitTransferFwdBwd,
                           controlNode := "Unit1.Em2.ControlNodes".cmSupportUnitTransferFwdBwd,
                           goToHomePos => "BA010AZCRPM01.11",
                           goToWorkPos => "BA010AZCRPM01.10");
END_REGION

REGION Network 98: CM Support Unit Shaft Up/Down Command Home
   RUNG wire#powerrail
      Contact( #TRUE )
      Coil( "Unit1.Em2.ControlNodes".cm.Interlock.SupportUnitShaft.home )
   END_RUNG
   RUNG wire#powerrail
      I_Contact( "Unit1.Em2.ControlNodes".SemiAutuSplice."step".action[311] )
      I_Contact( "Unit1.Em2.ControlNodes".SemiAutuSplice."step".action[411] )
      I_Contact( "Unit1.Em2.ControlNodes".SemiAutuSplice."step".action[414] )
      I_Contact( "Unit1.Em2.ControlNodes".SemiAutuSplice."step".action[1411] )
      I_Contact( "Unit1.Em2.ControlNodes".SemiAutuSplice."step".action[1511] )
      I_Contact( "Unit1.Em2.ControlNodes".SemiAutuSplice."step".action[2076] )
      Not()
      Contact( "Unit1.Em2.ControlNodes".cm.Interlock.SupportUnitShaft.home )
      Coil( "Unit1.Em2.ControlNodes".cmSupportUnitShaftUpDown.commands.commandHomePos )
   END_RUNG
   // the same network as SCL:
   "Unit1.Em2.ControlNodes".cm.Interlock.SupportUnitShaft.home := #TRUE;
   "Unit1.Em2.ControlNodes".cmSupportUnitShaftUpDown.commands.commandHomePos := NOT (NOT "Unit1.Em2.ControlNodes".SemiAutuSplice."step".action[311] AND NOT "Unit1.Em2.ControlNodes".SemiAutuSplice."step".action[411] AND NOT "Unit1.Em2.ControlNodes".SemiAutuSplice."step".action[414] AND NOT "Unit1.Em2.ControlNodes".SemiAutuSplice."step".action[1411] AND NOT "Unit1.Em2.ControlNodes".SemiAutuSplice."step".action[1511] AND NOT "Unit1.Em2.ControlNodes".SemiAutuSplice."step".action[2076]) AND "Unit1.Em2.ControlNodes".cm.Interlock.SupportUnitShaft.home;
END_REGION

REGION Network 99: CM Support Unit Shaft Up/Down Command Work
   RUNG wire#powerrail
      Contact( #TRUE )
      wire#w1
      Contact( "Unit1.Em2.ControlNodes".cmSupportUnitTransferFwdBwd.monitoring.inHomePos )
      wire#w2
      Coil( "Unit1.Em2.ControlNodes".cm.Interlock.SupportUnitShaft.work )
   END_RUNG
   RUNG wire#w1
      Contact( "Unit1.Em2.ControlNodes".cmSupportUnitTransferFwdBwd.monitoring.inWorkPos )
   END_RUNG wire#w2
   RUNG wire#powerrail
      I_Contact( "Unit1.Em2.ControlNodes".SemiAutuSplice."step".action[312] )
      I_Contact( "Unit1.Em2.ControlNodes".SemiAutuSplice."step".action[341] )
      I_Contact( "Unit1.Em2.ControlNodes".SemiAutuSplice."step".action[412] )
      I_Contact( "Unit1.Em2.ControlNodes".SemiAutuSplice."step".action[441] )
      I_Contact( "Unit1.Em2.ControlNodes".SemiAutuSplice."step".action[1431] )
      I_Contact( "Unit1.Em2.ControlNodes".SemiAutuSplice."step".action[1531] )
      I_Contact( "Unit1.Em2.ControlNodes".SemiAutuSplice."step".action[2088] )
      Not()
      Contact( "Unit1.Em2.ControlNodes".cm.Interlock.SupportUnitShaft.work )
      Coil( "Unit1.Em2.ControlNodes".cmSupportUnitShaftUpDown.commands.commandWorkPos )
   END_RUNG
   // the same network as SCL:
   "Unit1.Em2.ControlNodes".cm.Interlock.SupportUnitShaft.work := #TRUE AND ("Unit1.Em2.ControlNodes".cmSupportUnitTransferFwdBwd.monitoring.inHomePos OR "Unit1.Em2.ControlNodes".cmSupportUnitTransferFwdBwd.monitoring.inWorkPos);
   "Unit1.Em2.ControlNodes".cmSupportUnitShaftUpDown.commands.commandWorkPos := NOT (NOT "Unit1.Em2.ControlNodes".SemiAutuSplice."step".action[312] AND NOT "Unit1.Em2.ControlNodes".SemiAutuSplice."step".action[341] AND NOT "Unit1.Em2.ControlNodes".SemiAutuSplice."step".action[412] AND NOT "Unit1.Em2.ControlNodes".SemiAutuSplice."step".action[441] AND NOT "Unit1.Em2.ControlNodes".SemiAutuSplice."step".action[1431] AND NOT "Unit1.Em2.ControlNodes".SemiAutuSplice."step".action[1531] AND NOT "Unit1.Em2.ControlNodes".SemiAutuSplice."step".action[2088]) AND "Unit1.Em2.ControlNodes".cm.Interlock.SupportUnitShaft.work;
END_REGION

REGION Network 100: Call CM Support Unit Shaft Up/Down (LBC_TwoWayActuator)
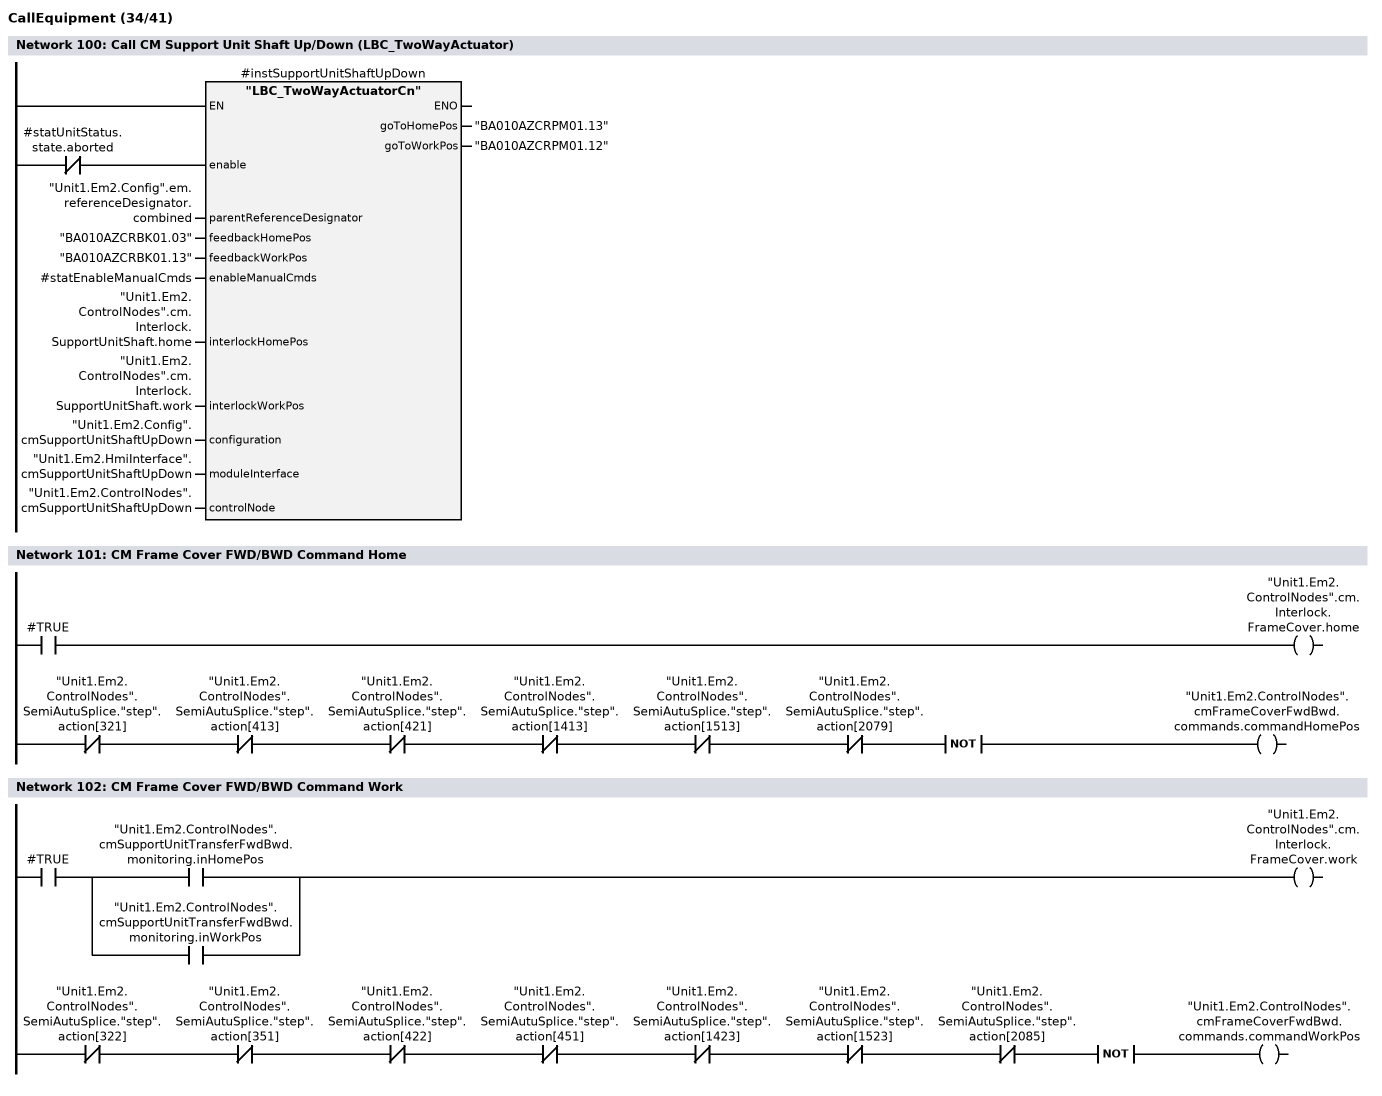
   RUNG wire#powerrail
      #instSupportUnitShaftUpDown(enable := wire#w1, parentReferenceDesignator := "Unit1.Em2.Config".em.referenceDesignator.combined, feedbackHomePos := "BA010AZCRBK01.03", feedbackWorkPos := "BA010AZCRBK01.13", enableManualCmds := #statEnableManualCmds, interlockHomePos := "Unit1.Em2.ControlNodes".cm.Interlock.SupportUnitShaft.home, interlockWorkPos := "Unit1.Em2.ControlNodes".cm.Interlock.SupportUnitShaft.work, configuration := "Unit1.Em2.Config".cmSupportUnitShaftUpDown, moduleInterface := "Unit1.Em2.HmiInterface".cmSupportUnitShaftUpDown, controlNode := "Unit1.Em2.ControlNodes".cmSupportUnitShaftUpDown, goToHomePos => "BA010AZCRPM01.13", goToWorkPos => "BA010AZCRPM01.12")
   END_RUNG
   RUNG wire#powerrail
      I_Contact( #statUnitStatus.state.aborted )
   END_RUNG wire#w1
   // the same network as SCL:
   #instSupportUnitShaftUpDown(enable := NOT #statUnitStatus.state.aborted,   // "LBC_TwoWayActuatorCn"
                           parentReferenceDesignator := "Unit1.Em2.Config".em.referenceDesignator.combined,
                           feedbackHomePos := "BA010AZCRBK01.03",
                           feedbackWorkPos := "BA010AZCRBK01.13",
                           enableManualCmds := #statEnableManualCmds,
                           interlockHomePos := "Unit1.Em2.ControlNodes".cm.Interlock.SupportUnitShaft.home,
                           interlockWorkPos := "Unit1.Em2.ControlNodes".cm.Interlock.SupportUnitShaft.work,
                           configuration := "Unit1.Em2.Config".cmSupportUnitShaftUpDown,
                           moduleInterface := "Unit1.Em2.HmiInterface".cmSupportUnitShaftUpDown,
                           controlNode := "Unit1.Em2.ControlNodes".cmSupportUnitShaftUpDown,
                           goToHomePos => "BA010AZCRPM01.13",
                           goToWorkPos => "BA010AZCRPM01.12");
END_REGION

REGION Network 101: CM Frame Cover FWD/BWD Command Home
   RUNG wire#powerrail
      Contact( #TRUE )
      Coil( "Unit1.Em2.ControlNodes".cm.Interlock.FrameCover.home )
   END_RUNG
   RUNG wire#powerrail
      I_Contact( "Unit1.Em2.ControlNodes".SemiAutuSplice."step".action[321] )
      I_Contact( "Unit1.Em2.ControlNodes".SemiAutuSplice."step".action[413] )
      I_Contact( "Unit1.Em2.ControlNodes".SemiAutuSplice."step".action[421] )
      I_Contact( "Unit1.Em2.ControlNodes".SemiAutuSplice."step".action[1413] )
      I_Contact( "Unit1.Em2.ControlNodes".SemiAutuSplice."step".action[1513] )
      I_Contact( "Unit1.Em2.ControlNodes".SemiAutuSplice."step".action[2079] )
      Not()
      Coil( "Unit1.Em2.ControlNodes".cmFrameCoverFwdBwd.commands.commandHomePos )
   END_RUNG
   // the same network as SCL:
   "Unit1.Em2.ControlNodes".cm.Interlock.FrameCover.home := #TRUE;
   "Unit1.Em2.ControlNodes".cmFrameCoverFwdBwd.commands.commandHomePos := NOT (NOT "Unit1.Em2.ControlNodes".SemiAutuSplice."step".action[321] AND NOT "Unit1.Em2.ControlNodes".SemiAutuSplice."step".action[413] AND NOT "Unit1.Em2.ControlNodes".SemiAutuSplice."step".action[421] AND NOT "Unit1.Em2.ControlNodes".SemiAutuSplice."step".action[1413] AND NOT "Unit1.Em2.ControlNodes".SemiAutuSplice."step".action[1513] AND NOT "Unit1.Em2.ControlNodes".SemiAutuSplice."step".action[2079]);
END_REGION

REGION Network 102: CM Frame Cover FWD/BWD Command Work
   RUNG wire#powerrail
      Contact( #TRUE )
      wire#w1
      Contact( "Unit1.Em2.ControlNodes".cmSupportUnitTransferFwdBwd.monitoring.inHomePos )
      wire#w2
      Coil( "Unit1.Em2.ControlNodes".cm.Interlock.FrameCover.work )
   END_RUNG
   RUNG wire#w1
      Contact( "Unit1.Em2.ControlNodes".cmSupportUnitTransferFwdBwd.monitoring.inWorkPos )
   END_RUNG wire#w2
   RUNG wire#powerrail
      I_Contact( "Unit1.Em2.ControlNodes".SemiAutuSplice."step".action[322] )
      I_Contact( "Unit1.Em2.ControlNodes".SemiAutuSplice."step".action[351] )
      I_Contact( "Unit1.Em2.ControlNodes".SemiAutuSplice."step".action[422] )
      I_Contact( "Unit1.Em2.ControlNodes".SemiAutuSplice."step".action[451] )
      I_Contact( "Unit1.Em2.ControlNodes".SemiAutuSplice."step".action[1423] )
      I_Contact( "Unit1.Em2.ControlNodes".SemiAutuSplice."step".action[1523] )
      I_Contact( "Unit1.Em2.ControlNodes".SemiAutuSplice."step".action[2085] )
      Not()
      Coil( "Unit1.Em2.ControlNodes".cmFrameCoverFwdBwd.commands.commandWorkPos )
   END_RUNG
   // the same network as SCL:
   "Unit1.Em2.ControlNodes".cm.Interlock.FrameCover.work := #TRUE AND ("Unit1.Em2.ControlNodes".cmSupportUnitTransferFwdBwd.monitoring.inHomePos OR "Unit1.Em2.ControlNodes".cmSupportUnitTransferFwdBwd.monitoring.inWorkPos);
   "Unit1.Em2.ControlNodes".cmFrameCoverFwdBwd.commands.commandWorkPos := NOT (NOT "Unit1.Em2.ControlNodes".SemiAutuSplice."step".action[322] AND NOT "Unit1.Em2.ControlNodes".SemiAutuSplice."step".action[351] AND NOT "Unit1.Em2.ControlNodes".SemiAutuSplice."step".action[422] AND NOT "Unit1.Em2.ControlNodes".SemiAutuSplice."step".action[451] AND NOT "Unit1.Em2.ControlNodes".SemiAutuSplice."step".action[1423] AND NOT "Unit1.Em2.ControlNodes".SemiAutuSplice."step".action[1523] AND NOT "Unit1.Em2.ControlNodes".SemiAutuSplice."step".action[2085]);
END_REGION

REGION Network 103: Call CM Frame Cover FWD/BWD (LBC_TwoWayActuator)
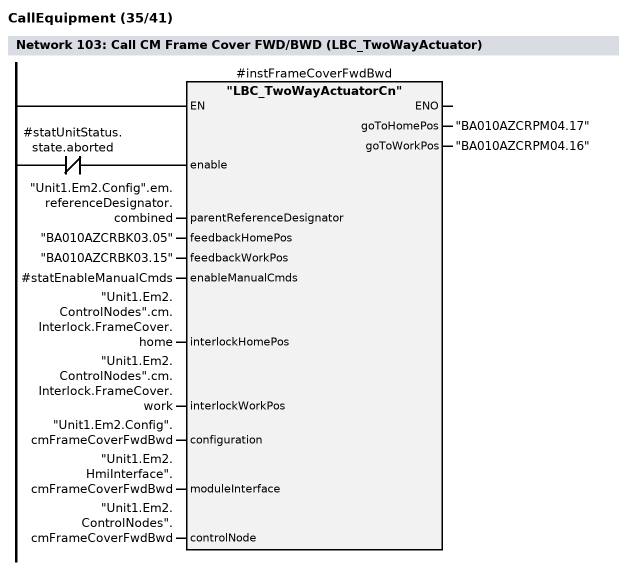
   RUNG wire#powerrail
      #instFrameCoverFwdBwd(enable := wire#w1, parentReferenceDesignator := "Unit1.Em2.Config".em.referenceDesignator.combined, feedbackHomePos := "BA010AZCRBK03.05", feedbackWorkPos := "BA010AZCRBK03.15", enableManualCmds := #statEnableManualCmds, interlockHomePos := "Unit1.Em2.ControlNodes".cm.Interlock.FrameCover.home, interlockWorkPos := "Unit1.Em2.ControlNodes".cm.Interlock.FrameCover.work, configuration := "Unit1.Em2.Config".cmFrameCoverFwdBwd, moduleInterface := "Unit1.Em2.HmiInterface".cmFrameCoverFwdBwd, controlNode := "Unit1.Em2.ControlNodes".cmFrameCoverFwdBwd, goToHomePos => "BA010AZCRPM04.17", goToWorkPos => "BA010AZCRPM04.16")
   END_RUNG
   RUNG wire#powerrail
      I_Contact( #statUnitStatus.state.aborted )
   END_RUNG wire#w1
   // the same network as SCL:
   #instFrameCoverFwdBwd(enable := NOT #statUnitStatus.state.aborted,   // "LBC_TwoWayActuatorCn"
                         parentReferenceDesignator := "Unit1.Em2.Config".em.referenceDesignator.combined,
                         feedbackHomePos := "BA010AZCRBK03.05",
                         feedbackWorkPos := "BA010AZCRBK03.15",
                         enableManualCmds := #statEnableManualCmds,
                         interlockHomePos := "Unit1.Em2.ControlNodes".cm.Interlock.FrameCover.home,
                         interlockWorkPos := "Unit1.Em2.ControlNodes".cm.Interlock.FrameCover.work,
                         configuration := "Unit1.Em2.Config".cmFrameCoverFwdBwd,
                         moduleInterface := "Unit1.Em2.HmiInterface".cmFrameCoverFwdBwd,
                         controlNode := "Unit1.Em2.ControlNodes".cmFrameCoverFwdBwd,
                         goToHomePos => "BA010AZCRPM04.17",
                         goToWorkPos => "BA010AZCRPM04.16");
END_REGION

REGION Network 104: ******************** Feedback to Unit ********************
END_REGION

REGION Network 105: Determine StateComplete (SC) in Mode Production
   // Conditions for the Equipment Modules "stateComplete" feedback to the unit. This feedback is given when the task in for the respective state is complete.
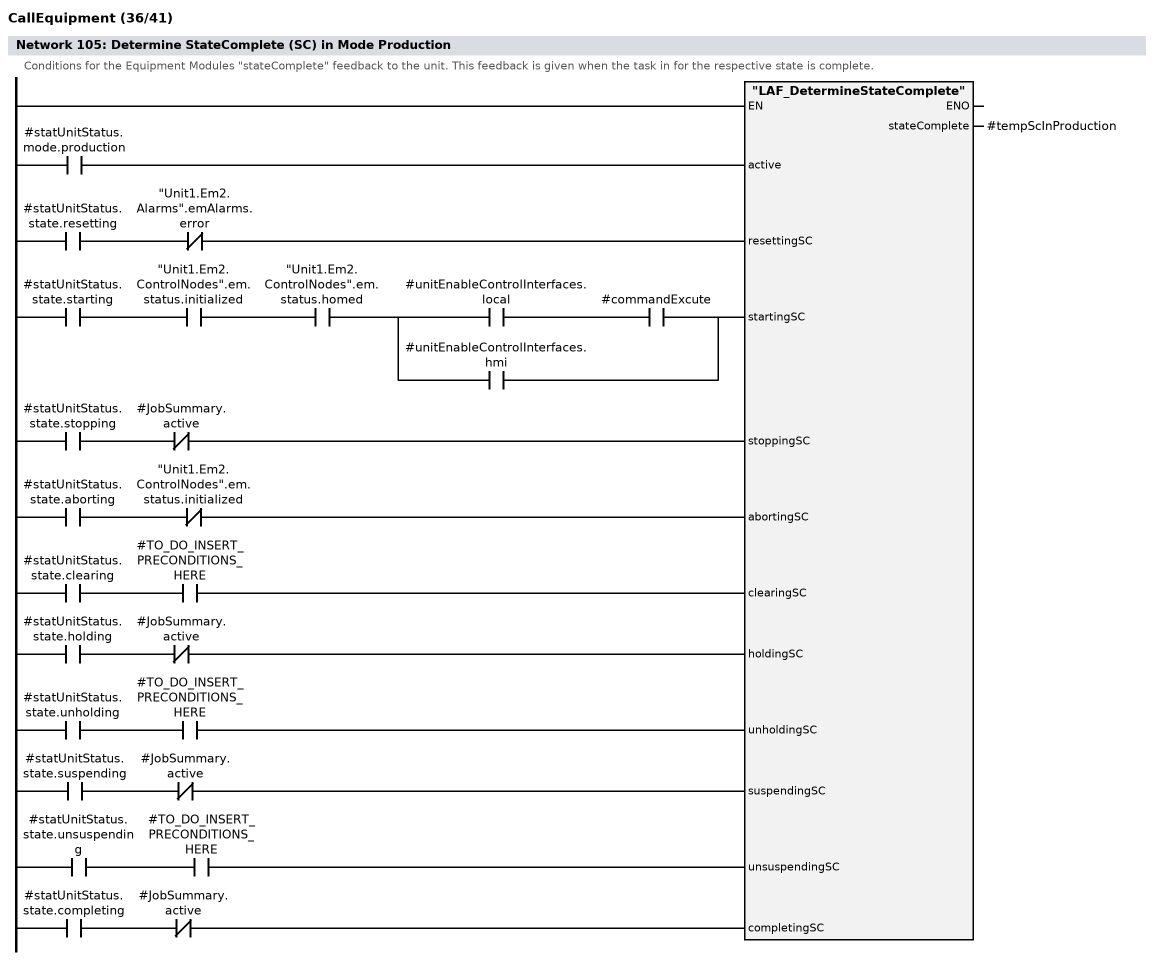
   RUNG wire#powerrail
      "LAF_DetermineStateComplete"(active := wire#w1, resettingSC := wire#w2, startingSC := wire#w4, stoppingSC := wire#w5, abortingSC := wire#w6, clearingSC := wire#w7, holdingSC := wire#w8, unholdingSC := wire#w9, suspendingSC := wire#w10, unsuspendingSC := wire#w11, completingSC := wire#w12, stateComplete => #tempScInProduction)
   END_RUNG
   RUNG wire#powerrail
      Contact( #statUnitStatus.mode.production )
   END_RUNG wire#w1
   RUNG wire#powerrail
      Contact( #statUnitStatus.state.resetting )
      I_Contact( "Unit1.Em2.Alarms".emAlarms.error )
   END_RUNG wire#w2
   RUNG wire#powerrail
      Contact( #statUnitStatus.state.starting )
      Contact( "Unit1.Em2.ControlNodes".em.status.initialized )
      Contact( "Unit1.Em2.ControlNodes".em.status.homed )
      wire#w3
      Contact( #unitEnableControlInterfaces.local )
      Contact( #commandExcute )
   END_RUNG wire#w4
   RUNG wire#w3
      Contact( #unitEnableControlInterfaces.hmi )
   END_RUNG wire#w4
   RUNG wire#powerrail
      Contact( #statUnitStatus.state.stopping )
      I_Contact( #JobSummary.active )
   END_RUNG wire#w5
   RUNG wire#powerrail
      Contact( #statUnitStatus.state.aborting )
      I_Contact( "Unit1.Em2.ControlNodes".em.status.initialized )
   END_RUNG wire#w6
   RUNG wire#powerrail
      Contact( #statUnitStatus.state.clearing )
      Contact( #TO_DO_INSERT_PRECONDITIONS_HERE )
   END_RUNG wire#w7
   RUNG wire#powerrail
      Contact( #statUnitStatus.state.holding )
      I_Contact( #JobSummary.active )
   END_RUNG wire#w8
   RUNG wire#powerrail
      Contact( #statUnitStatus.state.unholding )
      Contact( #TO_DO_INSERT_PRECONDITIONS_HERE )
   END_RUNG wire#w9
   RUNG wire#powerrail
      Contact( #statUnitStatus.state.suspending )
      I_Contact( #JobSummary.active )
   END_RUNG wire#w10
   RUNG wire#powerrail
      Contact( #statUnitStatus.state.unsuspending )
      Contact( #TO_DO_INSERT_PRECONDITIONS_HERE )
   END_RUNG wire#w11
   RUNG wire#powerrail
      Contact( #statUnitStatus.state.completing )
      I_Contact( #JobSummary.active )
   END_RUNG wire#w12
   // the same network as SCL:
   "LAF_DetermineStateComplete"(active := #statUnitStatus.mode.production,
                           resettingSC := #statUnitStatus.state.resetting AND NOT "Unit1.Em2.Alarms".emAlarms.error,
                           startingSC := #statUnitStatus.state.starting AND "Unit1.Em2.ControlNodes".em.status.initialized AND "Unit1.Em2.ControlNodes".em.status.homed AND ((#unitEnableControlInterfaces.local AND #commandExcute) OR #unitEnableControlInterfaces.hmi),
                           stoppingSC := #statUnitStatus.state.stopping AND NOT #JobSummary.active,
                           abortingSC := #statUnitStatus.state.aborting AND NOT "Unit1.Em2.ControlNodes".em.status.initialized,
                           clearingSC := #statUnitStatus.state.clearing AND #TO_DO_INSERT_PRECONDITIONS_HERE,
                           holdingSC := #statUnitStatus.state.holding AND NOT #JobSummary.active,
                           unholdingSC := #statUnitStatus.state.unholding AND #TO_DO_INSERT_PRECONDITIONS_HERE,
                           suspendingSC := #statUnitStatus.state.suspending AND NOT #JobSummary.active,
                           unsuspendingSC := #statUnitStatus.state.unsuspending AND #TO_DO_INSERT_PRECONDITIONS_HERE,
                           completingSC := #statUnitStatus.state.completing AND NOT #JobSummary.active,
                           stateComplete => #tempScInProduction);
END_REGION

REGION Network 106: Determine StateComplete (SC) in Mode Maintenance/Manual
   // Conditions for the Equipment Modules "stateComplete" feedback to the unit. This feedback is given when the task in for the respective state is complete.
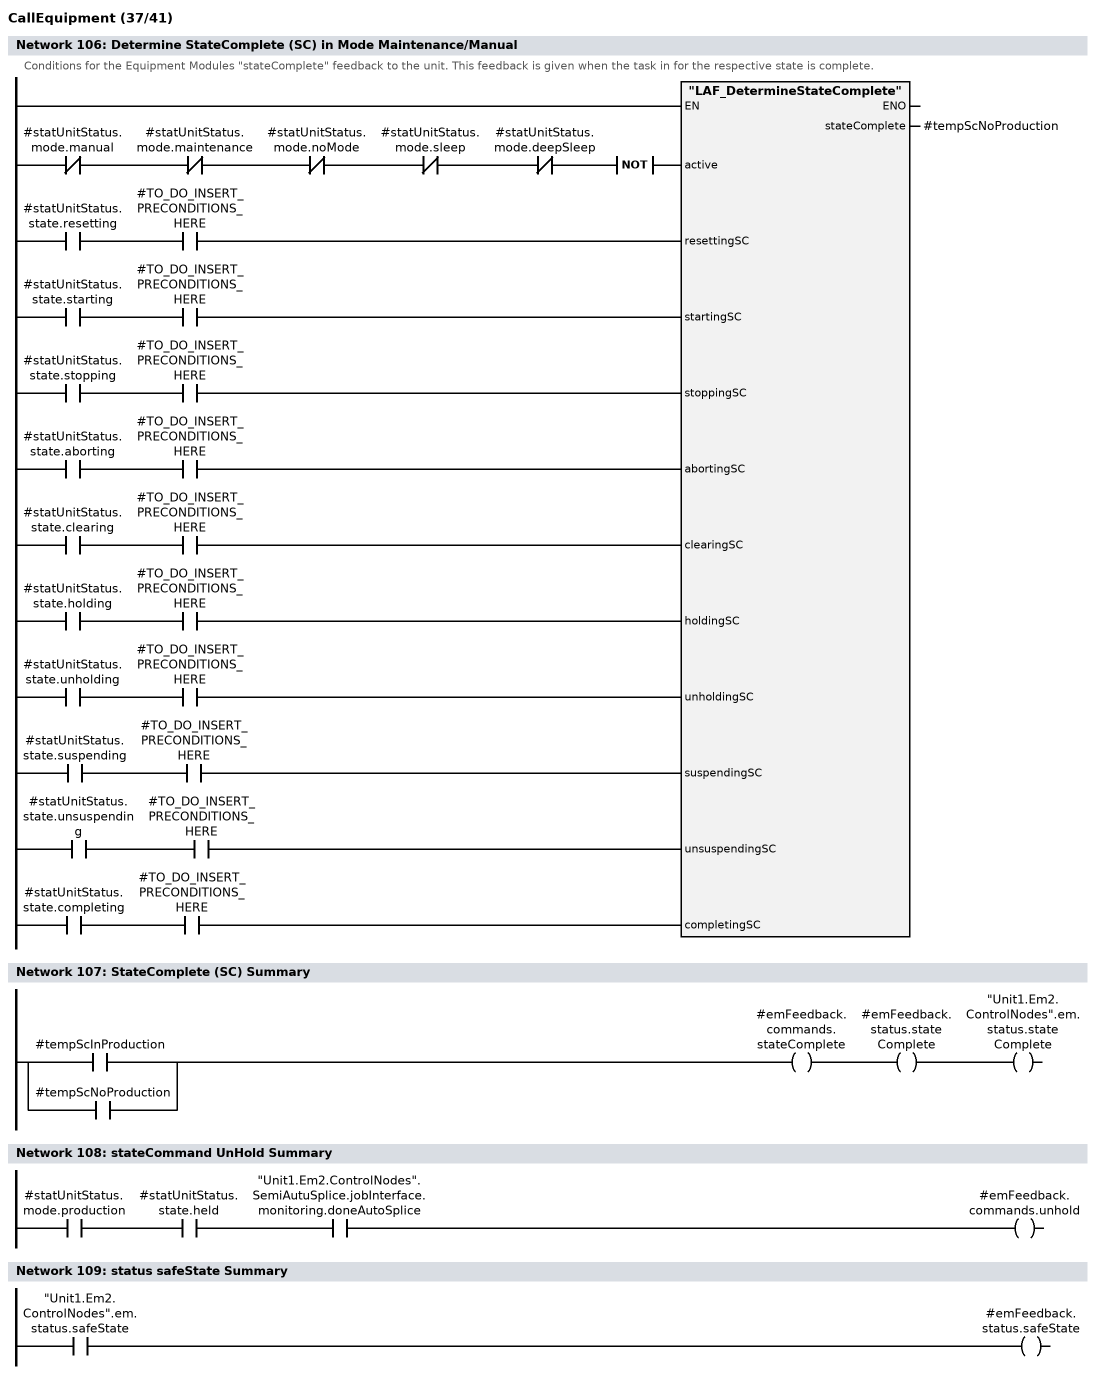
   RUNG wire#powerrail
      "LAF_DetermineStateComplete"(active := wire#w1, resettingSC := wire#w2, startingSC := wire#w3, stoppingSC := wire#w4, abortingSC := wire#w5, clearingSC := wire#w6, holdingSC := wire#w7, unholdingSC := wire#w8, suspendingSC := wire#w9, unsuspendingSC := wire#w10, completingSC := wire#w11, stateComplete => #tempScNoProduction)
   END_RUNG
   RUNG wire#powerrail
      I_Contact( #statUnitStatus.mode.manual )
      I_Contact( #statUnitStatus.mode.maintenance )
      I_Contact( #statUnitStatus.mode.noMode )
      I_Contact( #statUnitStatus.mode.sleep )
      I_Contact( #statUnitStatus.mode.deepSleep )
      Not()
   END_RUNG wire#w1
   RUNG wire#powerrail
      Contact( #statUnitStatus.state.resetting )
      Contact( #TO_DO_INSERT_PRECONDITIONS_HERE )
   END_RUNG wire#w2
   RUNG wire#powerrail
      Contact( #statUnitStatus.state.starting )
      Contact( #TO_DO_INSERT_PRECONDITIONS_HERE )
   END_RUNG wire#w3
   RUNG wire#powerrail
      Contact( #statUnitStatus.state.stopping )
      Contact( #TO_DO_INSERT_PRECONDITIONS_HERE )
   END_RUNG wire#w4
   RUNG wire#powerrail
      Contact( #statUnitStatus.state.aborting )
      Contact( #TO_DO_INSERT_PRECONDITIONS_HERE )
   END_RUNG wire#w5
   RUNG wire#powerrail
      Contact( #statUnitStatus.state.clearing )
      Contact( #TO_DO_INSERT_PRECONDITIONS_HERE )
   END_RUNG wire#w6
   RUNG wire#powerrail
      Contact( #statUnitStatus.state.holding )
      Contact( #TO_DO_INSERT_PRECONDITIONS_HERE )
   END_RUNG wire#w7
   RUNG wire#powerrail
      Contact( #statUnitStatus.state.unholding )
      Contact( #TO_DO_INSERT_PRECONDITIONS_HERE )
   END_RUNG wire#w8
   RUNG wire#powerrail
      Contact( #statUnitStatus.state.suspending )
      Contact( #TO_DO_INSERT_PRECONDITIONS_HERE )
   END_RUNG wire#w9
   RUNG wire#powerrail
      Contact( #statUnitStatus.state.unsuspending )
      Contact( #TO_DO_INSERT_PRECONDITIONS_HERE )
   END_RUNG wire#w10
   RUNG wire#powerrail
      Contact( #statUnitStatus.state.completing )
      Contact( #TO_DO_INSERT_PRECONDITIONS_HERE )
   END_RUNG wire#w11
   // the same network as SCL:
   "LAF_DetermineStateComplete"(active := NOT (NOT #statUnitStatus.mode.manual AND NOT #statUnitStatus.mode.maintenance AND NOT #statUnitStatus.mode.noMode AND NOT #statUnitStatus.mode.sleep AND NOT #statUnitStatus.mode.deepSleep),
                           resettingSC := #statUnitStatus.state.resetting AND #TO_DO_INSERT_PRECONDITIONS_HERE,
                           startingSC := #statUnitStatus.state.starting AND #TO_DO_INSERT_PRECONDITIONS_HERE,
                           stoppingSC := #statUnitStatus.state.stopping AND #TO_DO_INSERT_PRECONDITIONS_HERE,
                           abortingSC := #statUnitStatus.state.aborting AND #TO_DO_INSERT_PRECONDITIONS_HERE,
                           clearingSC := #statUnitStatus.state.clearing AND #TO_DO_INSERT_PRECONDITIONS_HERE,
                           holdingSC := #statUnitStatus.state.holding AND #TO_DO_INSERT_PRECONDITIONS_HERE,
                           unholdingSC := #statUnitStatus.state.unholding AND #TO_DO_INSERT_PRECONDITIONS_HERE,
                           suspendingSC := #statUnitStatus.state.suspending AND #TO_DO_INSERT_PRECONDITIONS_HERE,
                           unsuspendingSC := #statUnitStatus.state.unsuspending AND #TO_DO_INSERT_PRECONDITIONS_HERE,
                           completingSC := #statUnitStatus.state.completing AND #TO_DO_INSERT_PRECONDITIONS_HERE,
                           stateComplete => #tempScNoProduction);
END_REGION

REGION Network 107: StateComplete (SC) Summary
   RUNG wire#powerrail
      Contact( #tempScInProduction )
      wire#w1
      Coil( #emFeedback.commands.stateComplete )
      Coil( #emFeedback.status.stateComplete )
      Coil( "Unit1.Em2.ControlNodes".em.status.stateComplete )
   END_RUNG
   RUNG wire#powerrail
      Contact( #tempScNoProduction )
   END_RUNG wire#w1
   // the same network as SCL:
   #emFeedback.commands.stateComplete := #tempScInProduction OR #tempScNoProduction;
   #emFeedback.status.stateComplete := #emFeedback.commands.stateComplete;
   "Unit1.Em2.ControlNodes".em.status.stateComplete := #emFeedback.commands.stateComplete;
END_REGION

REGION Network 108: stateCommand UnHold Summary
   RUNG wire#powerrail
      Contact( #statUnitStatus.mode.production )
      Contact( #statUnitStatus.state.held )
      Contact( "Unit1.Em2.ControlNodes".SemiAutuSplice.jobInterface.monitoring.doneAutoSplice )
      Coil( #emFeedback.commands.unhold )
   END_RUNG
   // the same network as SCL:
   #emFeedback.commands.unhold := #statUnitStatus.mode.production AND #statUnitStatus.state.held AND "Unit1.Em2.ControlNodes".SemiAutuSplice.jobInterface.monitoring.doneAutoSplice;
END_REGION

REGION Network 109: status safeState Summary
   RUNG wire#powerrail
      Contact( "Unit1.Em2.ControlNodes".em.status.safeState )
      Coil( #emFeedback.status.safeState )
   END_RUNG
   // the same network as SCL:
   #emFeedback.status.safeState := "Unit1.Em2.ControlNodes".em.status.safeState;
END_REGION

REGION Network 110: status safetyReleased Summary
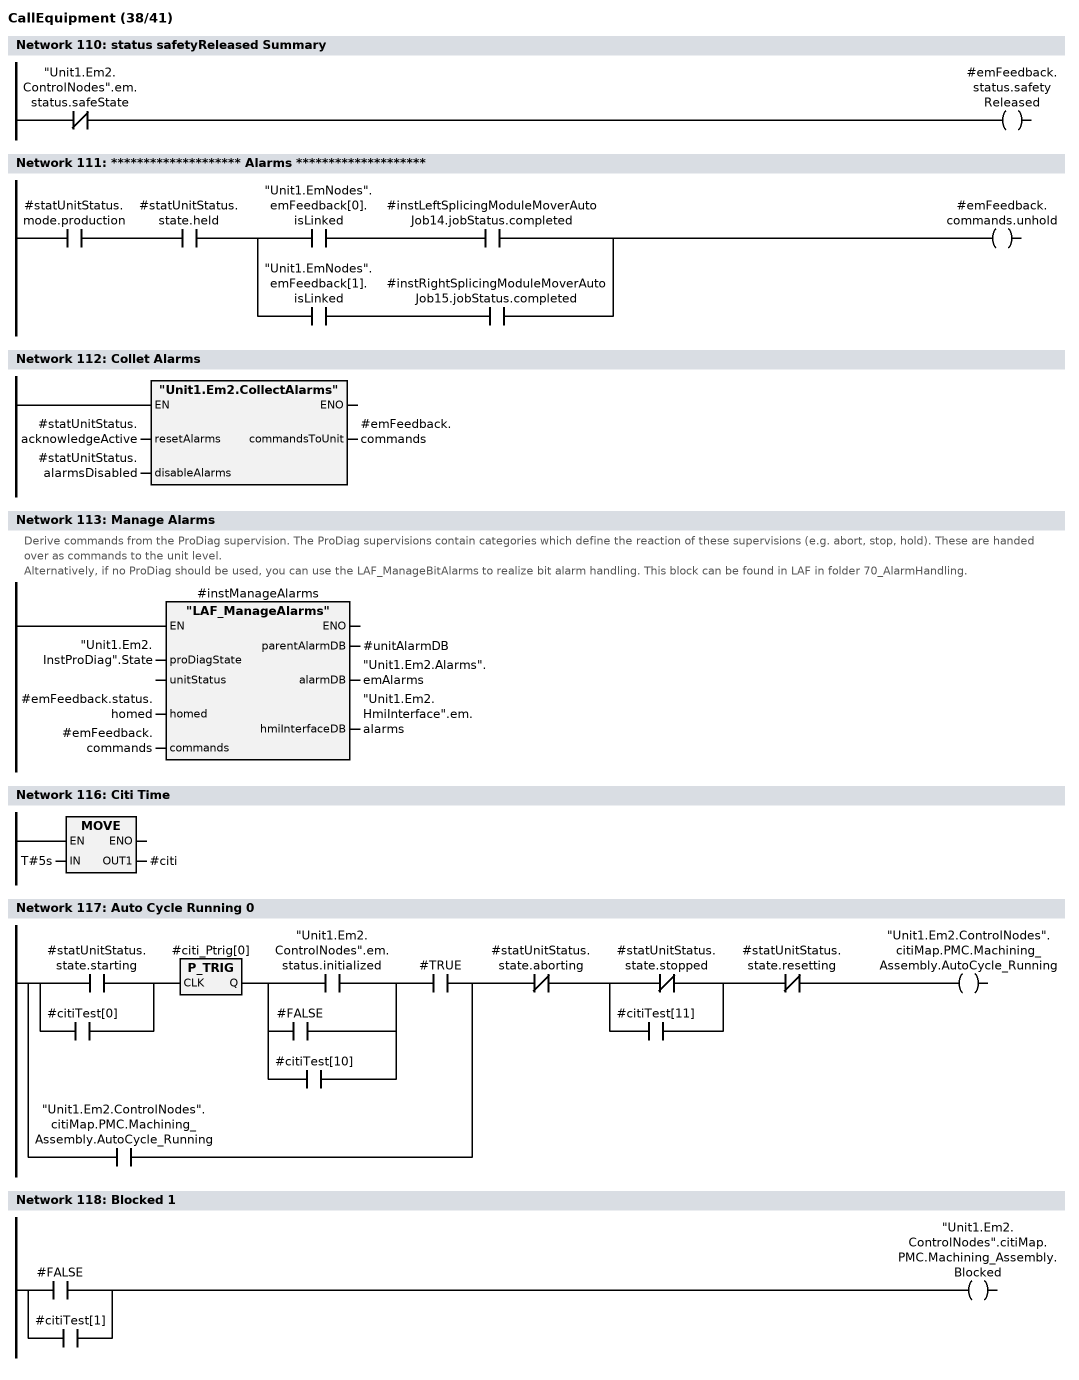
   RUNG wire#powerrail
      I_Contact( "Unit1.Em2.ControlNodes".em.status.safeState )
      Coil( #emFeedback.status.safetyReleased )
   END_RUNG
   // the same network as SCL:
   #emFeedback.status.safetyReleased := NOT "Unit1.Em2.ControlNodes".em.status.safeState;
END_REGION

REGION Network 111: ******************** Alarms ********************
   RUNG wire#powerrail
      Contact( #statUnitStatus.mode.production )
      Contact( #statUnitStatus.state.held )
      wire#w1
      Contact( "Unit1.EmNodes".emFeedback[0].isLinked )
      Contact( #instLeftSplicingModuleMoverAutoJob14.jobStatus.completed )
      wire#w2
      Coil( #emFeedback.commands.unhold )
   END_RUNG
   RUNG wire#w1
      Contact( "Unit1.EmNodes".emFeedback[1].isLinked )
      Contact( #instRightSplicingModuleMoverAutoJob15.jobStatus.completed )
   END_RUNG wire#w2
   // the same network as SCL:
   #emFeedback.commands.unhold := #statUnitStatus.mode.production AND #statUnitStatus.state.held AND (("Unit1.EmNodes".emFeedback[0].isLinked AND #instLeftSplicingModuleMoverAutoJob14.jobStatus.completed) OR ("Unit1.EmNodes".emFeedback[1].isLinked AND #instRightSplicingModuleMoverAutoJob15.jobStatus.completed));
END_REGION

REGION Network 112: Collet Alarms
   RUNG wire#powerrail
      "Unit1.Em2.CollectAlarms"(resetAlarms := #statUnitStatus.acknowledgeActive, disableAlarms := #statUnitStatus.alarmsDisabled, commandsToUnit => #emFeedback.commands)
   END_RUNG
   // the same network as SCL:
   "Unit1.Em2.CollectAlarms"(resetAlarms := #statUnitStatus.acknowledgeActive,
                           disableAlarms := #statUnitStatus.alarmsDisabled,
                           commandsToUnit => #emFeedback.commands);
END_REGION

REGION Network 113: Manage Alarms
   // Derive commands from the ProDiag supervision. The ProDiag supervisions contain categories which define the reaction of these supervisions (e.g. abort, stop, hold). These are handed over as commands to the unit level.
   // Alternatively, if no ProDiag should be used, you can use the LAF_ManageBitAlarms to realize bit alarm handling. This block can be found in LAF in folder 70_AlarmHandling.
   RUNG wire#powerrail
      #instManageAlarms(proDiagState := "Unit1.Em2.InstProDiag".State, homed := #emFeedback.status.homed, commands := #emFeedback.commands, parentAlarmDB => #unitAlarmDB, alarmDB => "Unit1.Em2.Alarms".emAlarms, hmiInterfaceDB => "Unit1.Em2.HmiInterface".em.alarms, unitStatus :=)
   END_RUNG
   // the same network as SCL:
   #instManageAlarms(proDiagState := "Unit1.Em2.InstProDiag".State,   // "LAF_ManageAlarms"
                     homed := #emFeedback.status.homed,
                     commands := #emFeedback.commands,
                     parentAlarmDB => #unitAlarmDB,
                     alarmDB => "Unit1.Em2.Alarms".emAlarms,
                     hmiInterfaceDB => "Unit1.Em2.HmiInterface".em.alarms);
END_REGION

REGION Network 115: ******************** CITI ********************
END_REGION

REGION Network 116: Citi Time
   RUNG wire#powerrail
      Move(in := T#5s, out1 => #citi)
   END_RUNG
   // the same network as SCL:
   #citi := T#5s;
END_REGION

REGION Network 117: Auto Cycle Running 0
   RUNG wire#powerrail
      Contact( #statUnitStatus.state.starting )
      wire#w1
      P_Trig( #citi_Ptrig[0] )
      wire#w2
      Contact( "Unit1.Em2.ControlNodes".em.status.initialized )
      wire#w3
      Contact( #TRUE )
      wire#w4
      I_Contact( #statUnitStatus.state.aborting )
      wire#w5
      I_Contact( #statUnitStatus.state.stopped )
      wire#w6
      I_Contact( #statUnitStatus.state.resetting )
      Coil( "Unit1.Em2.ControlNodes".citiMap.PMC.Machining_Assembly.AutoCycle_Running )
   END_RUNG
   RUNG wire#powerrail
      Contact( #citiTest[0] )
   END_RUNG wire#w1
   RUNG wire#w2
      Contact( #FALSE )
   END_RUNG wire#w3
   RUNG wire#w2
      Contact( #citiTest[10] )
   END_RUNG wire#w3
   RUNG wire#powerrail
      Contact( "Unit1.Em2.ControlNodes".citiMap.PMC.Machining_Assembly.AutoCycle_Running )
   END_RUNG wire#w4
   RUNG wire#w5
      Contact( #citiTest[11] )
   END_RUNG wire#w6
   // the same network as SCL:
   #_w1 := #statUnitStatus.state.starting OR #citiTest[0];
   #_w2 := #_w1 AND NOT #citi_Ptrig[0];   // rising edge
   #citi_Ptrig[0] := #_w1;
   "Unit1.Em2.ControlNodes".citiMap.PMC.Machining_Assembly.AutoCycle_Running := ((#_w2 AND ("Unit1.Em2.ControlNodes".em.status.initialized OR #FALSE OR #citiTest[10]) AND #TRUE) OR "Unit1.Em2.ControlNodes".citiMap.PMC.Machining_Assembly.AutoCycle_Running) AND NOT #statUnitStatus.state.aborting AND (NOT #statUnitStatus.state.stopped OR #citiTest[11]) AND NOT #statUnitStatus.state.resetting;
END_REGION

REGION Network 118: Blocked 1
   RUNG wire#powerrail
      Contact( #FALSE )
      wire#w1
      Coil( "Unit1.Em2.ControlNodes".citiMap.PMC.Machining_Assembly.Blocked )
   END_RUNG
   RUNG wire#powerrail
      Contact( #citiTest[1] )
   END_RUNG wire#w1
   // the same network as SCL:
   "Unit1.Em2.ControlNodes".citiMap.PMC.Machining_Assembly.Blocked := #FALSE OR #citiTest[1];
END_REGION

REGION Network 119: Starved 2
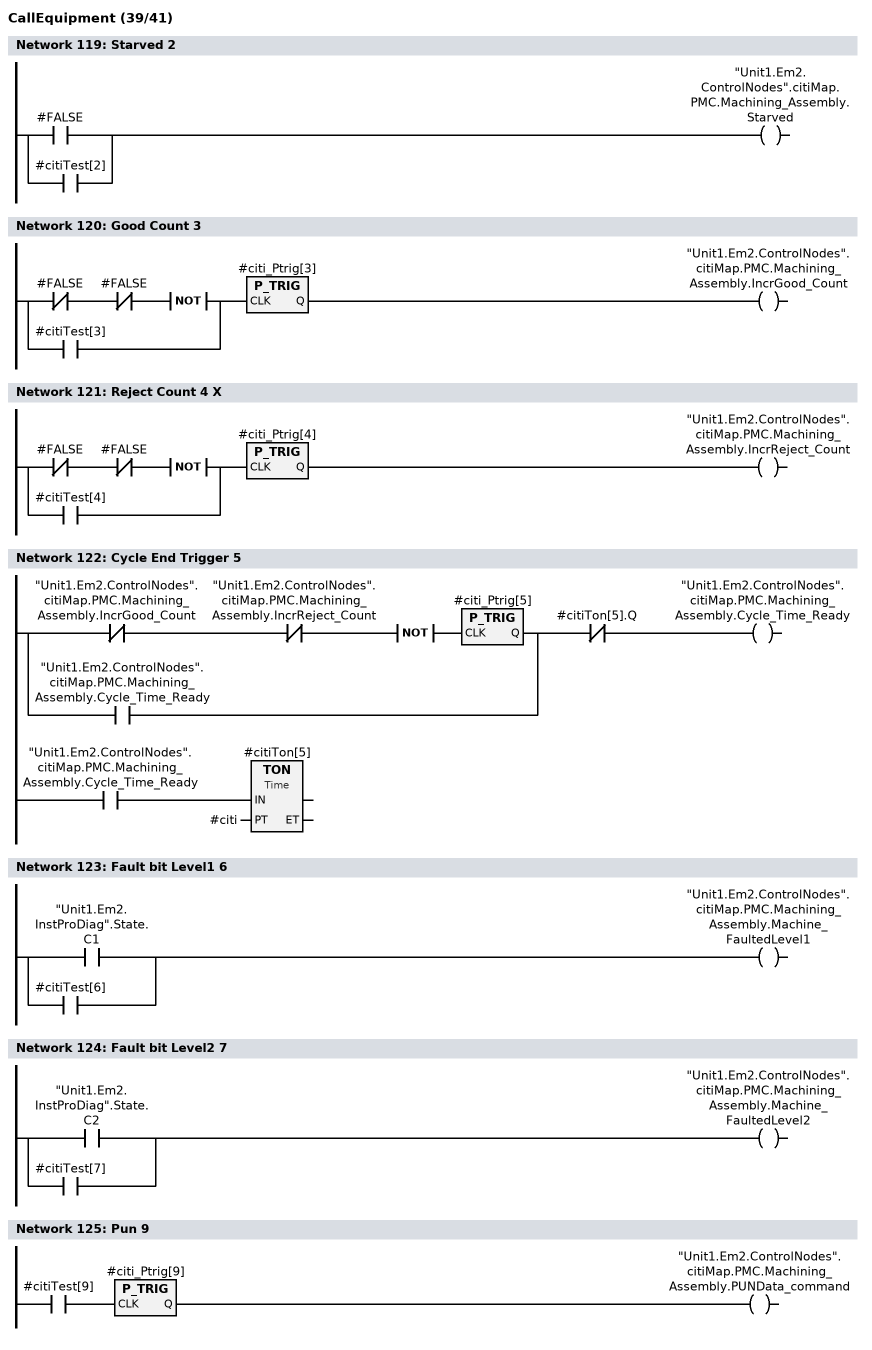
   RUNG wire#powerrail
      Contact( #FALSE )
      wire#w1
      Coil( "Unit1.Em2.ControlNodes".citiMap.PMC.Machining_Assembly.Starved )
   END_RUNG
   RUNG wire#powerrail
      Contact( #citiTest[2] )
   END_RUNG wire#w1
   // the same network as SCL:
   "Unit1.Em2.ControlNodes".citiMap.PMC.Machining_Assembly.Starved := #FALSE OR #citiTest[2];
END_REGION

REGION Network 120: Good Count 3
   RUNG wire#powerrail
      I_Contact( #FALSE )
      I_Contact( #FALSE )
      Not()
      wire#w1
      P_Trig( #citi_Ptrig[3] )
      Coil( "Unit1.Em2.ControlNodes".citiMap.PMC.Machining_Assembly.IncrGood_Count )
   END_RUNG
   RUNG wire#powerrail
      Contact( #citiTest[3] )
   END_RUNG wire#w1
   // the same network as SCL:
   #_w1 := NOT (NOT #FALSE AND NOT #FALSE) OR #citiTest[3];
   #_w2 := #_w1 AND NOT #citi_Ptrig[3];   // rising edge
   #citi_Ptrig[3] := #_w1;
   "Unit1.Em2.ControlNodes".citiMap.PMC.Machining_Assembly.IncrGood_Count := #_w2;
END_REGION

REGION Network 121: Reject Count 4 X
   RUNG wire#powerrail
      I_Contact( #FALSE )
      I_Contact( #FALSE )
      Not()
      wire#w1
      P_Trig( #citi_Ptrig[4] )
      Coil( "Unit1.Em2.ControlNodes".citiMap.PMC.Machining_Assembly.IncrReject_Count )
   END_RUNG
   RUNG wire#powerrail
      Contact( #citiTest[4] )
   END_RUNG wire#w1
   // the same network as SCL:
   #_w1 := NOT (NOT #FALSE AND NOT #FALSE) OR #citiTest[4];
   #_w2 := #_w1 AND NOT #citi_Ptrig[4];   // rising edge
   #citi_Ptrig[4] := #_w1;
   "Unit1.Em2.ControlNodes".citiMap.PMC.Machining_Assembly.IncrReject_Count := #_w2;
END_REGION

REGION Network 122: Cycle End Trigger 5
   RUNG wire#powerrail
      I_Contact( "Unit1.Em2.ControlNodes".citiMap.PMC.Machining_Assembly.IncrGood_Count )
      I_Contact( "Unit1.Em2.ControlNodes".citiMap.PMC.Machining_Assembly.IncrReject_Count )
      Not()
      P_Trig( #citi_Ptrig[5] )
      wire#w1
      I_Contact( #citiTon[5].Q )
      Coil( "Unit1.Em2.ControlNodes".citiMap.PMC.Machining_Assembly.Cycle_Time_Ready )
   END_RUNG
   RUNG wire#powerrail
      Contact( "Unit1.Em2.ControlNodes".citiMap.PMC.Machining_Assembly.Cycle_Time_Ready )
   END_RUNG wire#w1
   RUNG wire#powerrail
      Contact( "Unit1.Em2.ControlNodes".citiMap.PMC.Machining_Assembly.Cycle_Time_Ready )
      { S7_Templates := "time_type := Time" } #citiTon[5].TON(pt := #citi, et =>)
   END_RUNG
   // the same network as SCL:
   #_w1 := NOT (NOT "Unit1.Em2.ControlNodes".citiMap.PMC.Machining_Assembly.IncrGood_Count AND NOT "Unit1.Em2.ControlNodes".citiMap.PMC.Machining_Assembly.IncrReject_Count);
   #_w2 := #_w1 AND NOT #citi_Ptrig[5];   // rising edge
   #citi_Ptrig[5] := #_w1;
   "Unit1.Em2.ControlNodes".citiMap.PMC.Machining_Assembly.Cycle_Time_Ready := (#_w2 OR "Unit1.Em2.ControlNodes".citiMap.PMC.Machining_Assembly.Cycle_Time_Ready) AND NOT #citiTon[5].Q;
   #citiTon[5].TON(IN := "Unit1.Em2.ControlNodes".citiMap.PMC.Machining_Assembly.Cycle_Time_Ready, PT := #citi);
END_REGION

REGION Network 123: Fault bit Level1 6
   RUNG wire#powerrail
      Contact( "Unit1.Em2.InstProDiag".State.C1 )
      wire#w1
      Coil( "Unit1.Em2.ControlNodes".citiMap.PMC.Machining_Assembly.Machine_FaultedLevel1 )
   END_RUNG
   RUNG wire#powerrail
      Contact( #citiTest[6] )
   END_RUNG wire#w1
   // the same network as SCL:
   "Unit1.Em2.ControlNodes".citiMap.PMC.Machining_Assembly.Machine_FaultedLevel1 := "Unit1.Em2.InstProDiag".State.C1 OR #citiTest[6];
END_REGION

REGION Network 124: Fault bit Level2 7
   RUNG wire#powerrail
      Contact( "Unit1.Em2.InstProDiag".State.C2 )
      wire#w1
      Coil( "Unit1.Em2.ControlNodes".citiMap.PMC.Machining_Assembly.Machine_FaultedLevel2 )
   END_RUNG
   RUNG wire#powerrail
      Contact( #citiTest[7] )
   END_RUNG wire#w1
   // the same network as SCL:
   "Unit1.Em2.ControlNodes".citiMap.PMC.Machining_Assembly.Machine_FaultedLevel2 := "Unit1.Em2.InstProDiag".State.C2 OR #citiTest[7];
END_REGION

REGION Network 125: Pun 9
   RUNG wire#powerrail
      Contact( #citiTest[9] )
      P_Trig( #citi_Ptrig[9] )
      Coil( "Unit1.Em2.ControlNodes".citiMap.PMC.Machining_Assembly.PUNData_command )
   END_RUNG
   // the same network as SCL:
   #_w1 := #citiTest[9] AND NOT #citi_Ptrig[9];   // rising edge
   #citi_Ptrig[9] := #citiTest[9];
   "Unit1.Em2.ControlNodes".citiMap.PMC.Machining_Assembly.PUNData_command := #_w1;
END_REGION

REGION Network 126: ControlNodes.CitiMap -> Unit1. EmNodes.emIt01
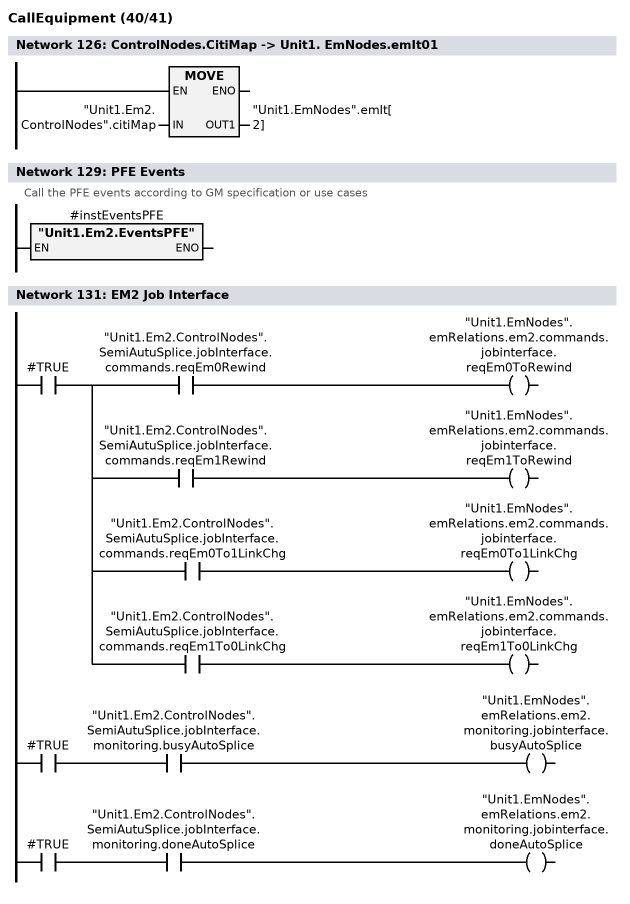
   RUNG wire#powerrail
      Move(in := "Unit1.Em2.ControlNodes".citiMap, out1 => "Unit1.EmNodes".emIt[2])
   END_RUNG
   // the same network as SCL:
   "Unit1.EmNodes".emIt[2] := "Unit1.Em2.ControlNodes".citiMap;
END_REGION

REGION Network 128: ******************** PFE Events ********************
END_REGION

REGION Network 129: PFE Events
   // Call the PFE events according to GM specification or use cases
   RUNG wire#powerrail
      #instEventsPFE()
   END_RUNG
   // the same network as SCL:
   #instEventsPFE();   // "Unit1.Em2.EventsPFE"
END_REGION

REGION Network 130: ******************** EM Relations Output ********************
END_REGION

REGION Network 131: EM2 Job Interface
   RUNG wire#powerrail
      Contact( #TRUE )
      wire#w1
      Contact( "Unit1.Em2.ControlNodes".SemiAutuSplice.jobInterface.commands.reqEm0Rewind )
      Coil( "Unit1.EmNodes".emRelations.em2.commands.jobinterface.reqEm0ToRewind )
   END_RUNG
   RUNG wire#w1
      Contact( "Unit1.Em2.ControlNodes".SemiAutuSplice.jobInterface.commands.reqEm1Rewind )
      Coil( "Unit1.EmNodes".emRelations.em2.commands.jobinterface.reqEm1ToRewind )
   END_RUNG
   RUNG wire#w1
      Contact( "Unit1.Em2.ControlNodes".SemiAutuSplice.jobInterface.commands.reqEm0To1LinkChg )
      Coil( "Unit1.EmNodes".emRelations.em2.commands.jobinterface.reqEm0To1LinkChg )
   END_RUNG
   RUNG wire#w1
      Contact( "Unit1.Em2.ControlNodes".SemiAutuSplice.jobInterface.commands.reqEm1To0LinkChg )
      Coil( "Unit1.EmNodes".emRelations.em2.commands.jobinterface.reqEm1To0LinkChg )
   END_RUNG
   RUNG wire#powerrail
      Contact( #TRUE )
      Contact( "Unit1.Em2.ControlNodes".SemiAutuSplice.jobInterface.monitoring.busyAutoSplice )
      Coil( "Unit1.EmNodes".emRelations.em2.monitoring.jobinterface.busyAutoSplice )
   END_RUNG
   RUNG wire#powerrail
      Contact( #TRUE )
      Contact( "Unit1.Em2.ControlNodes".SemiAutuSplice.jobInterface.monitoring.doneAutoSplice )
      Coil( "Unit1.EmNodes".emRelations.em2.monitoring.jobinterface.doneAutoSplice )
   END_RUNG
   // the same network as SCL:
   "Unit1.EmNodes".emRelations.em2.commands.jobinterface.reqEm0ToRewind := #TRUE AND "Unit1.Em2.ControlNodes".SemiAutuSplice.jobInterface.commands.reqEm0Rewind;
   "Unit1.EmNodes".emRelations.em2.commands.jobinterface.reqEm1ToRewind := #TRUE AND "Unit1.Em2.ControlNodes".SemiAutuSplice.jobInterface.commands.reqEm1Rewind;
   "Unit1.EmNodes".emRelations.em2.commands.jobinterface.reqEm0To1LinkChg := #TRUE AND "Unit1.Em2.ControlNodes".SemiAutuSplice.jobInterface.commands.reqEm0To1LinkChg;
   "Unit1.EmNodes".emRelations.em2.commands.jobinterface.reqEm1To0LinkChg := #TRUE AND "Unit1.Em2.ControlNodes".SemiAutuSplice.jobInterface.commands.reqEm1To0LinkChg;
   "Unit1.EmNodes".emRelations.em2.monitoring.jobinterface.busyAutoSplice := #TRUE AND "Unit1.Em2.ControlNodes".SemiAutuSplice.jobInterface.monitoring.busyAutoSplice;
   "Unit1.EmNodes".emRelations.em2.monitoring.jobinterface.doneAutoSplice := #TRUE AND "Unit1.Em2.ControlNodes".SemiAutuSplice.jobInterface.monitoring.doneAutoSplice;
END_REGION

